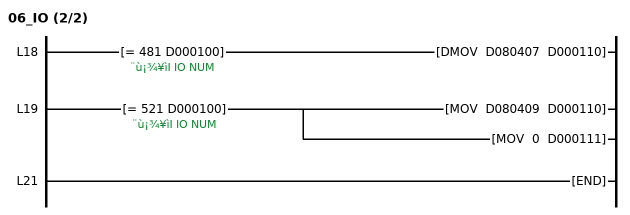
[picture p48: 06_IO rungs L18-L21]
; L18
LOAD=     481 D000100	// ¨ù¡¾¥ìI IO NUM
DMOV      D080407 D000110
; L19
LOAD=     521 D000100	// ¨ù¡¾¥ìI IO NUM
MOV       D080409 D000110
MOV       0 D000111
; L21
END

PROGRAM 07_VACUUM (task: ¨ö¨¬A¥ì CA¡¤I¡¾¡¿¡¤¡Í)

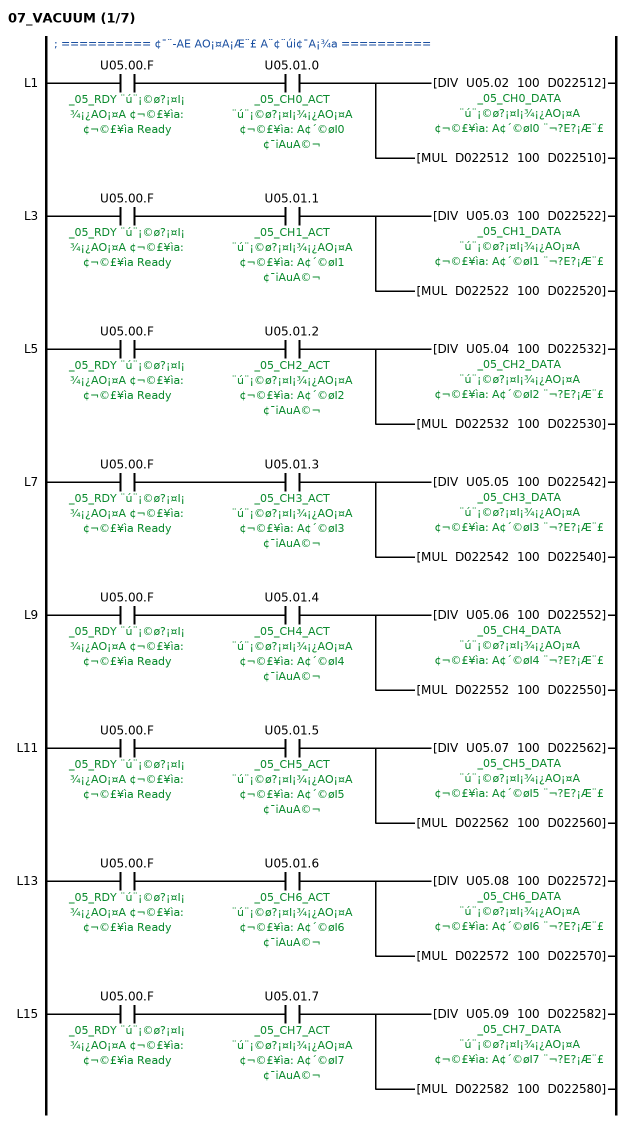
// ========== ¢¯¨­AE AO¡¤A¡Æ¨£ A¨¢¨úi¢¯A¡¾a ==========
; L1
LOAD      U05.00.F	// _05_RDY ¨ú¨¡©ø?¡¤I¡¾¡¿AO¡¤A ¢¬©£¥ìa: ¢¬©£¥ìa Ready
AND       U05.01.0	// _05_CH0_ACT ¨ú¨¡©ø?¡¤I¡¾¡¿AO¡¤A ¢¬©£¥ìa: A¢´©øI0 ¢¯iAuA©¬
DIV       U05.02 100 D022512	// _05_CH0_DATA ¨ú¨¡©ø?¡¤I¡¾¡¿AO¡¤A ¢¬©£¥ìa: A¢´©øI0 ¨¬?E?¡Æ¨£
MUL       D022512 100 D022510
; L3
LOAD      U05.00.F	// _05_RDY ¨ú¨¡©ø?¡¤I¡¾¡¿AO¡¤A ¢¬©£¥ìa: ¢¬©£¥ìa Ready
AND       U05.01.1	// _05_CH1_ACT ¨ú¨¡©ø?¡¤I¡¾¡¿AO¡¤A ¢¬©£¥ìa: A¢´©øI1 ¢¯iAuA©¬
DIV       U05.03 100 D022522	// _05_CH1_DATA ¨ú¨¡©ø?¡¤I¡¾¡¿AO¡¤A ¢¬©£¥ìa: A¢´©øI1 ¨¬?E?¡Æ¨£
MUL       D022522 100 D022520
; L5
LOAD      U05.00.F	// _05_RDY ¨ú¨¡©ø?¡¤I¡¾¡¿AO¡¤A ¢¬©£¥ìa: ¢¬©£¥ìa Ready
AND       U05.01.2	// _05_CH2_ACT ¨ú¨¡©ø?¡¤I¡¾¡¿AO¡¤A ¢¬©£¥ìa: A¢´©øI2 ¢¯iAuA©¬
DIV       U05.04 100 D022532	// _05_CH2_DATA ¨ú¨¡©ø?¡¤I¡¾¡¿AO¡¤A ¢¬©£¥ìa: A¢´©øI2 ¨¬?E?¡Æ¨£
MUL       D022532 100 D022530
; L7
LOAD      U05.00.F	// _05_RDY ¨ú¨¡©ø?¡¤I¡¾¡¿AO¡¤A ¢¬©£¥ìa: ¢¬©£¥ìa Ready
AND       U05.01.3	// _05_CH3_ACT ¨ú¨¡©ø?¡¤I¡¾¡¿AO¡¤A ¢¬©£¥ìa: A¢´©øI3 ¢¯iAuA©¬
DIV       U05.05 100 D022542	// _05_CH3_DATA ¨ú¨¡©ø?¡¤I¡¾¡¿AO¡¤A ¢¬©£¥ìa: A¢´©øI3 ¨¬?E?¡Æ¨£
MUL       D022542 100 D022540
; L9
LOAD      U05.00.F	// _05_RDY ¨ú¨¡©ø?¡¤I¡¾¡¿AO¡¤A ¢¬©£¥ìa: ¢¬©£¥ìa Ready
AND       U05.01.4	// _05_CH4_ACT ¨ú¨¡©ø?¡¤I¡¾¡¿AO¡¤A ¢¬©£¥ìa: A¢´©øI4 ¢¯iAuA©¬
DIV       U05.06 100 D022552	// _05_CH4_DATA ¨ú¨¡©ø?¡¤I¡¾¡¿AO¡¤A ¢¬©£¥ìa: A¢´©øI4 ¨¬?E?¡Æ¨£
MUL       D022552 100 D022550
; L11
LOAD      U05.00.F	// _05_RDY ¨ú¨¡©ø?¡¤I¡¾¡¿AO¡¤A ¢¬©£¥ìa: ¢¬©£¥ìa Ready
AND       U05.01.5	// _05_CH5_ACT ¨ú¨¡©ø?¡¤I¡¾¡¿AO¡¤A ¢¬©£¥ìa: A¢´©øI5 ¢¯iAuA©¬
DIV       U05.07 100 D022562	// _05_CH5_DATA ¨ú¨¡©ø?¡¤I¡¾¡¿AO¡¤A ¢¬©£¥ìa: A¢´©øI5 ¨¬?E?¡Æ¨£
MUL       D022562 100 D022560
; L13
LOAD      U05.00.F	// _05_RDY ¨ú¨¡©ø?¡¤I¡¾¡¿AO¡¤A ¢¬©£¥ìa: ¢¬©£¥ìa Ready
AND       U05.01.6	// _05_CH6_ACT ¨ú¨¡©ø?¡¤I¡¾¡¿AO¡¤A ¢¬©£¥ìa: A¢´©øI6 ¢¯iAuA©¬
DIV       U05.08 100 D022572	// _05_CH6_DATA ¨ú¨¡©ø?¡¤I¡¾¡¿AO¡¤A ¢¬©£¥ìa: A¢´©øI6 ¨¬?E?¡Æ¨£
MUL       D022572 100 D022570
; L15
LOAD      U05.00.F	// _05_RDY ¨ú¨¡©ø?¡¤I¡¾¡¿AO¡¤A ¢¬©£¥ìa: ¢¬©£¥ìa Ready
AND       U05.01.7	// _05_CH7_ACT ¨ú¨¡©ø?¡¤I¡¾¡¿AO¡¤A ¢¬©£¥ìa: A¢´©øI7 ¢¯iAuA©¬
DIV       U05.09 100 D022582	// _05_CH7_DATA ¨ú¨¡©ø?¡¤I¡¾¡¿AO¡¤A ¢¬©£¥ìa: A¢´©øI7 ¨¬?E?¡Æ¨£
MUL       D022582 100 D022580

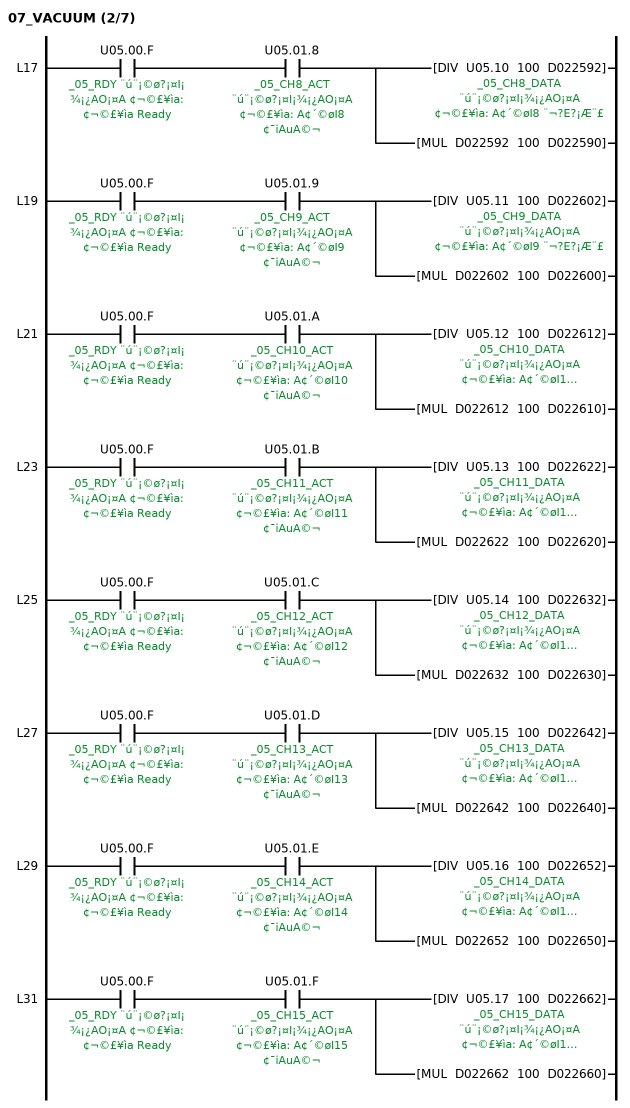
; L17
LOAD      U05.00.F	// _05_RDY ¨ú¨¡©ø?¡¤I¡¾¡¿AO¡¤A ¢¬©£¥ìa: ¢¬©£¥ìa Ready
AND       U05.01.8	// _05_CH8_ACT ¨ú¨¡©ø?¡¤I¡¾¡¿AO¡¤A ¢¬©£¥ìa: A¢´©øI8 ¢¯iAuA©¬
DIV       U05.10 100 D022592	// _05_CH8_DATA ¨ú¨¡©ø?¡¤I¡¾¡¿AO¡¤A ¢¬©£¥ìa: A¢´©øI8 ¨¬?E?¡Æ¨£
MUL       D022592 100 D022590
; L19
LOAD      U05.00.F	// _05_RDY ¨ú¨¡©ø?¡¤I¡¾¡¿AO¡¤A ¢¬©£¥ìa: ¢¬©£¥ìa Ready
AND       U05.01.9	// _05_CH9_ACT ¨ú¨¡©ø?¡¤I¡¾¡¿AO¡¤A ¢¬©£¥ìa: A¢´©øI9 ¢¯iAuA©¬
DIV       U05.11 100 D022602	// _05_CH9_DATA ¨ú¨¡©ø?¡¤I¡¾¡¿AO¡¤A ¢¬©£¥ìa: A¢´©øI9 ¨¬?E?¡Æ¨£
MUL       D022602 100 D022600
; L21
LOAD      U05.00.F	// _05_RDY ¨ú¨¡©ø?¡¤I¡¾¡¿AO¡¤A ¢¬©£¥ìa: ¢¬©£¥ìa Ready
AND       U05.01.A	// _05_CH10_ACT ¨ú¨¡©ø?¡¤I¡¾¡¿AO¡¤A ¢¬©£¥ìa: A¢´©øI10 ¢¯iAuA©¬
DIV       U05.12 100 D022612	// _05_CH10_DATA ¨ú¨¡©ø?¡¤I¡¾¡¿AO¡¤A ¢¬©£¥ìa: A¢´©øI10 ¨¬?E?¡Æ¨£
MUL       D022612 100 D022610
; L23
LOAD      U05.00.F	// _05_RDY ¨ú¨¡©ø?¡¤I¡¾¡¿AO¡¤A ¢¬©£¥ìa: ¢¬©£¥ìa Ready
AND       U05.01.B	// _05_CH11_ACT ¨ú¨¡©ø?¡¤I¡¾¡¿AO¡¤A ¢¬©£¥ìa: A¢´©øI11 ¢¯iAuA©¬
DIV       U05.13 100 D022622	// _05_CH11_DATA ¨ú¨¡©ø?¡¤I¡¾¡¿AO¡¤A ¢¬©£¥ìa: A¢´©øI11 ¨¬?E?¡Æ¨£
MUL       D022622 100 D022620
; L25
LOAD      U05.00.F	// _05_RDY ¨ú¨¡©ø?¡¤I¡¾¡¿AO¡¤A ¢¬©£¥ìa: ¢¬©£¥ìa Ready
AND       U05.01.C	// _05_CH12_ACT ¨ú¨¡©ø?¡¤I¡¾¡¿AO¡¤A ¢¬©£¥ìa: A¢´©øI12 ¢¯iAuA©¬
DIV       U05.14 100 D022632	// _05_CH12_DATA ¨ú¨¡©ø?¡¤I¡¾¡¿AO¡¤A ¢¬©£¥ìa: A¢´©øI12 ¨¬?E?¡Æ¨£
MUL       D022632 100 D022630
; L27
LOAD      U05.00.F	// _05_RDY ¨ú¨¡©ø?¡¤I¡¾¡¿AO¡¤A ¢¬©£¥ìa: ¢¬©£¥ìa Ready
AND       U05.01.D	// _05_CH13_ACT ¨ú¨¡©ø?¡¤I¡¾¡¿AO¡¤A ¢¬©£¥ìa: A¢´©øI13 ¢¯iAuA©¬
DIV       U05.15 100 D022642	// _05_CH13_DATA ¨ú¨¡©ø?¡¤I¡¾¡¿AO¡¤A ¢¬©£¥ìa: A¢´©øI13 ¨¬?E?¡Æ¨£
MUL       D022642 100 D022640
; L29
LOAD      U05.00.F	// _05_RDY ¨ú¨¡©ø?¡¤I¡¾¡¿AO¡¤A ¢¬©£¥ìa: ¢¬©£¥ìa Ready
AND       U05.01.E	// _05_CH14_ACT ¨ú¨¡©ø?¡¤I¡¾¡¿AO¡¤A ¢¬©£¥ìa: A¢´©øI14 ¢¯iAuA©¬
DIV       U05.16 100 D022652	// _05_CH14_DATA ¨ú¨¡©ø?¡¤I¡¾¡¿AO¡¤A ¢¬©£¥ìa: A¢´©øI14 ¨¬?E?¡Æ¨£
MUL       D022652 100 D022650
; L31
LOAD      U05.00.F	// _05_RDY ¨ú¨¡©ø?¡¤I¡¾¡¿AO¡¤A ¢¬©£¥ìa: ¢¬©£¥ìa Ready
AND       U05.01.F	// _05_CH15_ACT ¨ú¨¡©ø?¡¤I¡¾¡¿AO¡¤A ¢¬©£¥ìa: A¢´©øI15 ¢¯iAuA©¬
DIV       U05.17 100 D022662	// _05_CH15_DATA ¨ú¨¡©ø?¡¤I¡¾¡¿AO¡¤A ¢¬©£¥ìa: A¢´©øI15 ¨¬?E?¡Æ¨£
MUL       D022662 100 D022660

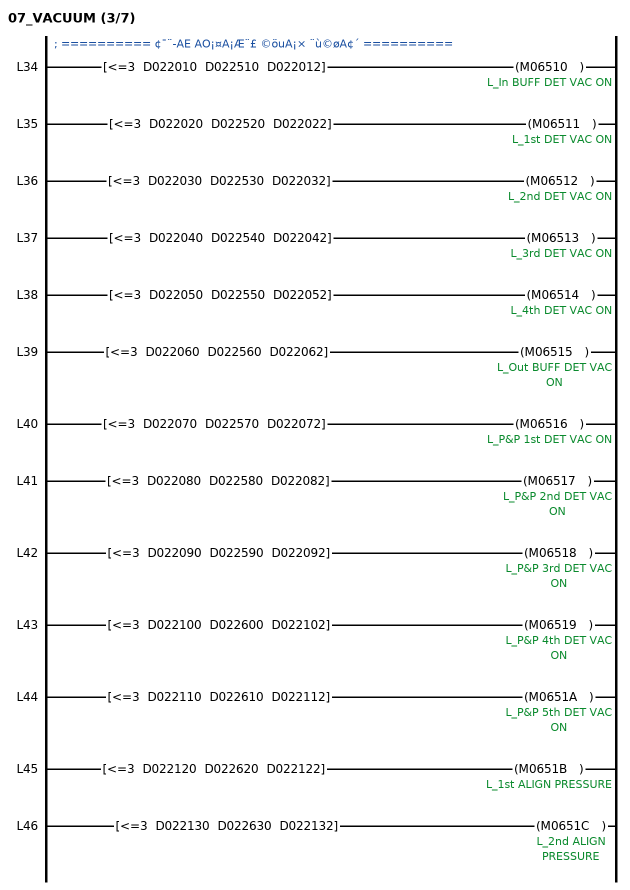
// ========== ¢¯¨­AE AO¡¤A¡Æ¨£ ©öuA¡× ¨ù©øA¢´ ==========
; L34
LOAD<=3   D022010 D022510 D022012
OUT       M06510	// L_In BUFF DET VAC ON
; L35
LOAD<=3   D022020 D022520 D022022
OUT       M06511	// L_1st DET VAC ON
; L36
LOAD<=3   D022030 D022530 D022032
OUT       M06512	// L_2nd DET VAC ON
; L37
LOAD<=3   D022040 D022540 D022042
OUT       M06513	// L_3rd DET VAC ON
; L38
LOAD<=3   D022050 D022550 D022052
OUT       M06514	// L_4th DET VAC ON
; L39
LOAD<=3   D022060 D022560 D022062
OUT       M06515	// L_Out BUFF DET VAC ON
; L40
LOAD<=3   D022070 D022570 D022072
OUT       M06516	// L_P&P 1st DET VAC ON
; L41
LOAD<=3   D022080 D022580 D022082
OUT       M06517	// L_P&P 2nd DET VAC ON
; L42
LOAD<=3   D022090 D022590 D022092
OUT       M06518	// L_P&P 3rd DET VAC ON
; L43
LOAD<=3   D022100 D022600 D022102
OUT       M06519	// L_P&P 4th DET VAC ON
; L44
LOAD<=3   D022110 D022610 D022112
OUT       M0651A	// L_P&P 5th DET VAC ON
; L45
LOAD<=3   D022120 D022620 D022122
OUT       M0651B	// L_1st ALIGN PRESSURE
; L46
LOAD<=3   D022130 D022630 D022132
OUT       M0651C	// L_2nd ALIGN PRESSURE

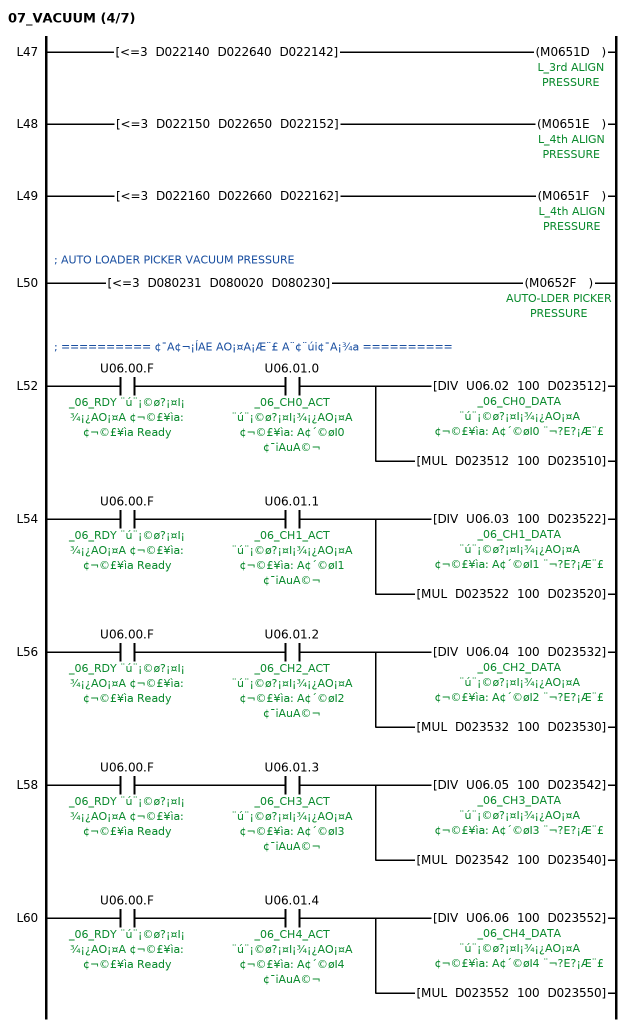
; L47
LOAD<=3   D022140 D022640 D022142
OUT       M0651D	// L_3rd ALIGN PRESSURE
; L48
LOAD<=3   D022150 D022650 D022152
OUT       M0651E	// L_4th ALIGN PRESSURE
; L49
LOAD<=3   D022160 D022660 D022162
OUT       M0651F	// L_4th ALIGN PRESSURE
; L50
LOAD<=3   D080231 D080020 D080230
OUT       M0652F	// AUTO-LDER PICKER PRESSURE
// output comment: AUTO LOADER PICKER VACUUM PRESSURE
// ========== ¢¯A¢¬¡ÍAE AO¡¤A¡Æ¨£ A¨¢¨úi¢¯A¡¾a ==========
; L52
LOAD      U06.00.F	// _06_RDY ¨ú¨¡©ø?¡¤I¡¾¡¿AO¡¤A ¢¬©£¥ìa: ¢¬©£¥ìa Ready
AND       U06.01.0	// _06_CH0_ACT ¨ú¨¡©ø?¡¤I¡¾¡¿AO¡¤A ¢¬©£¥ìa: A¢´©øI0 ¢¯iAuA©¬
DIV       U06.02 100 D023512	// _06_CH0_DATA ¨ú¨¡©ø?¡¤I¡¾¡¿AO¡¤A ¢¬©£¥ìa: A¢´©øI0 ¨¬?E?¡Æ¨£
MUL       D023512 100 D023510
; L54
LOAD      U06.00.F	// _06_RDY ¨ú¨¡©ø?¡¤I¡¾¡¿AO¡¤A ¢¬©£¥ìa: ¢¬©£¥ìa Ready
AND       U06.01.1	// _06_CH1_ACT ¨ú¨¡©ø?¡¤I¡¾¡¿AO¡¤A ¢¬©£¥ìa: A¢´©øI1 ¢¯iAuA©¬
DIV       U06.03 100 D023522	// _06_CH1_DATA ¨ú¨¡©ø?¡¤I¡¾¡¿AO¡¤A ¢¬©£¥ìa: A¢´©øI1 ¨¬?E?¡Æ¨£
MUL       D023522 100 D023520
; L56
LOAD      U06.00.F	// _06_RDY ¨ú¨¡©ø?¡¤I¡¾¡¿AO¡¤A ¢¬©£¥ìa: ¢¬©£¥ìa Ready
AND       U06.01.2	// _06_CH2_ACT ¨ú¨¡©ø?¡¤I¡¾¡¿AO¡¤A ¢¬©£¥ìa: A¢´©øI2 ¢¯iAuA©¬
DIV       U06.04 100 D023532	// _06_CH2_DATA ¨ú¨¡©ø?¡¤I¡¾¡¿AO¡¤A ¢¬©£¥ìa: A¢´©øI2 ¨¬?E?¡Æ¨£
MUL       D023532 100 D023530
; L58
LOAD      U06.00.F	// _06_RDY ¨ú¨¡©ø?¡¤I¡¾¡¿AO¡¤A ¢¬©£¥ìa: ¢¬©£¥ìa Ready
AND       U06.01.3	// _06_CH3_ACT ¨ú¨¡©ø?¡¤I¡¾¡¿AO¡¤A ¢¬©£¥ìa: A¢´©øI3 ¢¯iAuA©¬
DIV       U06.05 100 D023542	// _06_CH3_DATA ¨ú¨¡©ø?¡¤I¡¾¡¿AO¡¤A ¢¬©£¥ìa: A¢´©øI3 ¨¬?E?¡Æ¨£
MUL       D023542 100 D023540
; L60
LOAD      U06.00.F	// _06_RDY ¨ú¨¡©ø?¡¤I¡¾¡¿AO¡¤A ¢¬©£¥ìa: ¢¬©£¥ìa Ready
AND       U06.01.4	// _06_CH4_ACT ¨ú¨¡©ø?¡¤I¡¾¡¿AO¡¤A ¢¬©£¥ìa: A¢´©øI4 ¢¯iAuA©¬
DIV       U06.06 100 D023552	// _06_CH4_DATA ¨ú¨¡©ø?¡¤I¡¾¡¿AO¡¤A ¢¬©£¥ìa: A¢´©øI4 ¨¬?E?¡Æ¨£
MUL       D023552 100 D023550

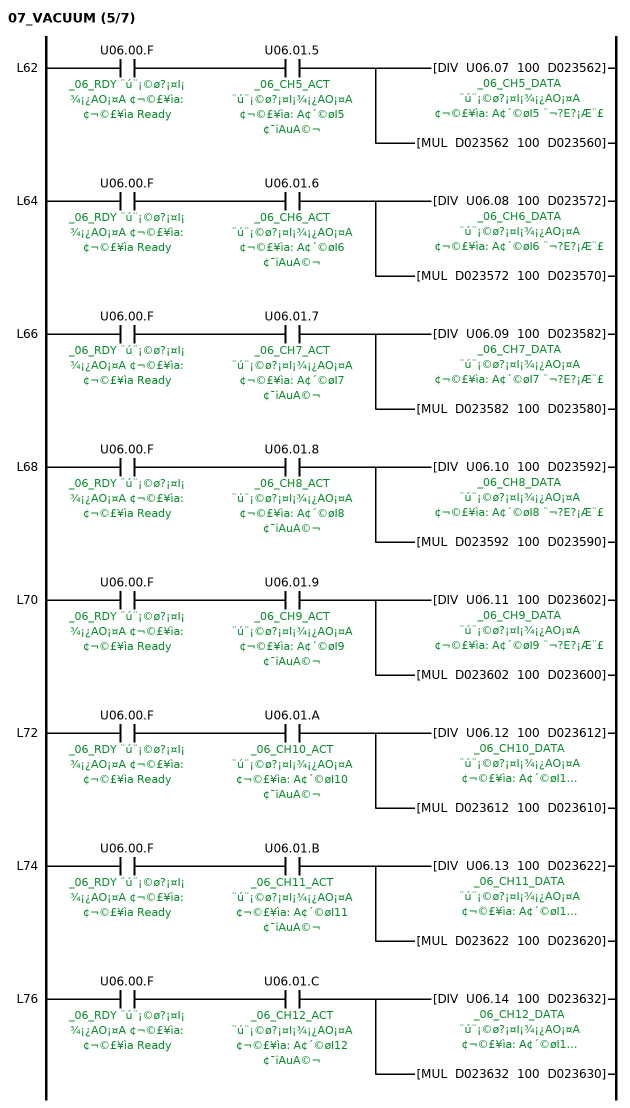
; L62
LOAD      U06.00.F	// _06_RDY ¨ú¨¡©ø?¡¤I¡¾¡¿AO¡¤A ¢¬©£¥ìa: ¢¬©£¥ìa Ready
AND       U06.01.5	// _06_CH5_ACT ¨ú¨¡©ø?¡¤I¡¾¡¿AO¡¤A ¢¬©£¥ìa: A¢´©øI5 ¢¯iAuA©¬
DIV       U06.07 100 D023562	// _06_CH5_DATA ¨ú¨¡©ø?¡¤I¡¾¡¿AO¡¤A ¢¬©£¥ìa: A¢´©øI5 ¨¬?E?¡Æ¨£
MUL       D023562 100 D023560
; L64
LOAD      U06.00.F	// _06_RDY ¨ú¨¡©ø?¡¤I¡¾¡¿AO¡¤A ¢¬©£¥ìa: ¢¬©£¥ìa Ready
AND       U06.01.6	// _06_CH6_ACT ¨ú¨¡©ø?¡¤I¡¾¡¿AO¡¤A ¢¬©£¥ìa: A¢´©øI6 ¢¯iAuA©¬
DIV       U06.08 100 D023572	// _06_CH6_DATA ¨ú¨¡©ø?¡¤I¡¾¡¿AO¡¤A ¢¬©£¥ìa: A¢´©øI6 ¨¬?E?¡Æ¨£
MUL       D023572 100 D023570
; L66
LOAD      U06.00.F	// _06_RDY ¨ú¨¡©ø?¡¤I¡¾¡¿AO¡¤A ¢¬©£¥ìa: ¢¬©£¥ìa Ready
AND       U06.01.7	// _06_CH7_ACT ¨ú¨¡©ø?¡¤I¡¾¡¿AO¡¤A ¢¬©£¥ìa: A¢´©øI7 ¢¯iAuA©¬
DIV       U06.09 100 D023582	// _06_CH7_DATA ¨ú¨¡©ø?¡¤I¡¾¡¿AO¡¤A ¢¬©£¥ìa: A¢´©øI7 ¨¬?E?¡Æ¨£
MUL       D023582 100 D023580
; L68
LOAD      U06.00.F	// _06_RDY ¨ú¨¡©ø?¡¤I¡¾¡¿AO¡¤A ¢¬©£¥ìa: ¢¬©£¥ìa Ready
AND       U06.01.8	// _06_CH8_ACT ¨ú¨¡©ø?¡¤I¡¾¡¿AO¡¤A ¢¬©£¥ìa: A¢´©øI8 ¢¯iAuA©¬
DIV       U06.10 100 D023592	// _06_CH8_DATA ¨ú¨¡©ø?¡¤I¡¾¡¿AO¡¤A ¢¬©£¥ìa: A¢´©øI8 ¨¬?E?¡Æ¨£
MUL       D023592 100 D023590
; L70
LOAD      U06.00.F	// _06_RDY ¨ú¨¡©ø?¡¤I¡¾¡¿AO¡¤A ¢¬©£¥ìa: ¢¬©£¥ìa Ready
AND       U06.01.9	// _06_CH9_ACT ¨ú¨¡©ø?¡¤I¡¾¡¿AO¡¤A ¢¬©£¥ìa: A¢´©øI9 ¢¯iAuA©¬
DIV       U06.11 100 D023602	// _06_CH9_DATA ¨ú¨¡©ø?¡¤I¡¾¡¿AO¡¤A ¢¬©£¥ìa: A¢´©øI9 ¨¬?E?¡Æ¨£
MUL       D023602 100 D023600
; L72
LOAD      U06.00.F	// _06_RDY ¨ú¨¡©ø?¡¤I¡¾¡¿AO¡¤A ¢¬©£¥ìa: ¢¬©£¥ìa Ready
AND       U06.01.A	// _06_CH10_ACT ¨ú¨¡©ø?¡¤I¡¾¡¿AO¡¤A ¢¬©£¥ìa: A¢´©øI10 ¢¯iAuA©¬
DIV       U06.12 100 D023612	// _06_CH10_DATA ¨ú¨¡©ø?¡¤I¡¾¡¿AO¡¤A ¢¬©£¥ìa: A¢´©øI10 ¨¬?E?¡Æ¨£
MUL       D023612 100 D023610
; L74
LOAD      U06.00.F	// _06_RDY ¨ú¨¡©ø?¡¤I¡¾¡¿AO¡¤A ¢¬©£¥ìa: ¢¬©£¥ìa Ready
AND       U06.01.B	// _06_CH11_ACT ¨ú¨¡©ø?¡¤I¡¾¡¿AO¡¤A ¢¬©£¥ìa: A¢´©øI11 ¢¯iAuA©¬
DIV       U06.13 100 D023622	// _06_CH11_DATA ¨ú¨¡©ø?¡¤I¡¾¡¿AO¡¤A ¢¬©£¥ìa: A¢´©øI11 ¨¬?E?¡Æ¨£
MUL       D023622 100 D023620
; L76
LOAD      U06.00.F	// _06_RDY ¨ú¨¡©ø?¡¤I¡¾¡¿AO¡¤A ¢¬©£¥ìa: ¢¬©£¥ìa Ready
AND       U06.01.C	// _06_CH12_ACT ¨ú¨¡©ø?¡¤I¡¾¡¿AO¡¤A ¢¬©£¥ìa: A¢´©øI12 ¢¯iAuA©¬
DIV       U06.14 100 D023632	// _06_CH12_DATA ¨ú¨¡©ø?¡¤I¡¾¡¿AO¡¤A ¢¬©£¥ìa: A¢´©øI12 ¨¬?E?¡Æ¨£
MUL       D023632 100 D023630

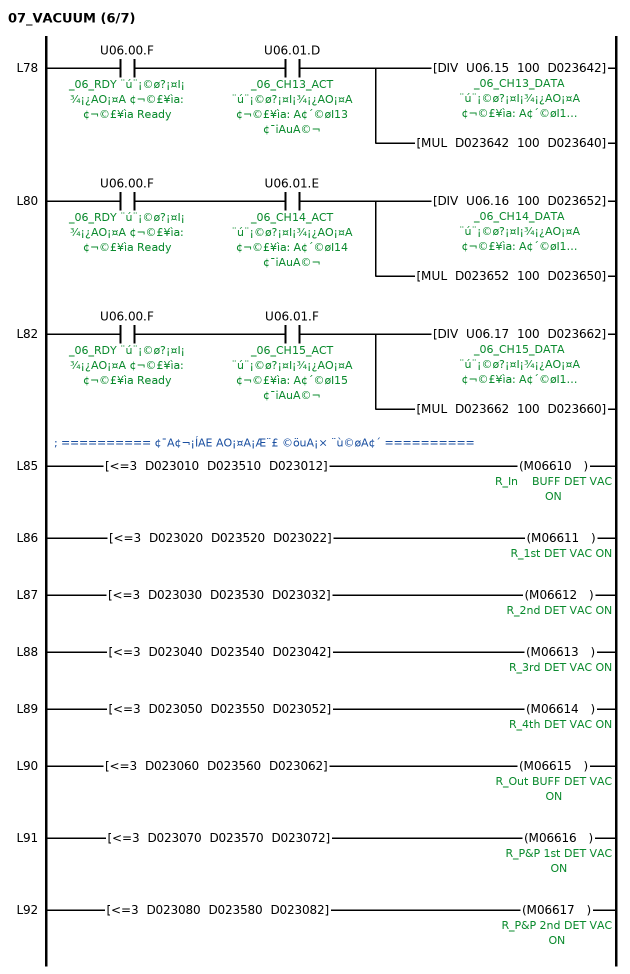
; L78
LOAD      U06.00.F	// _06_RDY ¨ú¨¡©ø?¡¤I¡¾¡¿AO¡¤A ¢¬©£¥ìa: ¢¬©£¥ìa Ready
AND       U06.01.D	// _06_CH13_ACT ¨ú¨¡©ø?¡¤I¡¾¡¿AO¡¤A ¢¬©£¥ìa: A¢´©øI13 ¢¯iAuA©¬
DIV       U06.15 100 D023642	// _06_CH13_DATA ¨ú¨¡©ø?¡¤I¡¾¡¿AO¡¤A ¢¬©£¥ìa: A¢´©øI13 ¨¬?E?¡Æ¨£
MUL       D023642 100 D023640
; L80
LOAD      U06.00.F	// _06_RDY ¨ú¨¡©ø?¡¤I¡¾¡¿AO¡¤A ¢¬©£¥ìa: ¢¬©£¥ìa Ready
AND       U06.01.E	// _06_CH14_ACT ¨ú¨¡©ø?¡¤I¡¾¡¿AO¡¤A ¢¬©£¥ìa: A¢´©øI14 ¢¯iAuA©¬
DIV       U06.16 100 D023652	// _06_CH14_DATA ¨ú¨¡©ø?¡¤I¡¾¡¿AO¡¤A ¢¬©£¥ìa: A¢´©øI14 ¨¬?E?¡Æ¨£
MUL       D023652 100 D023650
; L82
LOAD      U06.00.F	// _06_RDY ¨ú¨¡©ø?¡¤I¡¾¡¿AO¡¤A ¢¬©£¥ìa: ¢¬©£¥ìa Ready
AND       U06.01.F	// _06_CH15_ACT ¨ú¨¡©ø?¡¤I¡¾¡¿AO¡¤A ¢¬©£¥ìa: A¢´©øI15 ¢¯iAuA©¬
DIV       U06.17 100 D023662	// _06_CH15_DATA ¨ú¨¡©ø?¡¤I¡¾¡¿AO¡¤A ¢¬©£¥ìa: A¢´©øI15 ¨¬?E?¡Æ¨£
MUL       D023662 100 D023660
// ========== ¢¯A¢¬¡ÍAE AO¡¤A¡Æ¨£ ©öuA¡× ¨ù©øA¢´ ==========
; L85
LOAD<=3   D023010 D023510 D023012
OUT       M06610	// R_In    BUFF DET VAC ON
; L86
LOAD<=3   D023020 D023520 D023022
OUT       M06611	// R_1st DET VAC ON
; L87
LOAD<=3   D023030 D023530 D023032
OUT       M06612	// R_2nd DET VAC ON
; L88
LOAD<=3   D023040 D023540 D023042
OUT       M06613	// R_3rd DET VAC ON
; L89
LOAD<=3   D023050 D023550 D023052
OUT       M06614	// R_4th DET VAC ON
; L90
LOAD<=3   D023060 D023560 D023062
OUT       M06615	// R_Out BUFF DET VAC ON
; L91
LOAD<=3   D023070 D023570 D023072
OUT       M06616	// R_P&P 1st DET VAC ON
; L92
LOAD<=3   D023080 D023580 D023082
OUT       M06617	// R_P&P 2nd DET VAC ON

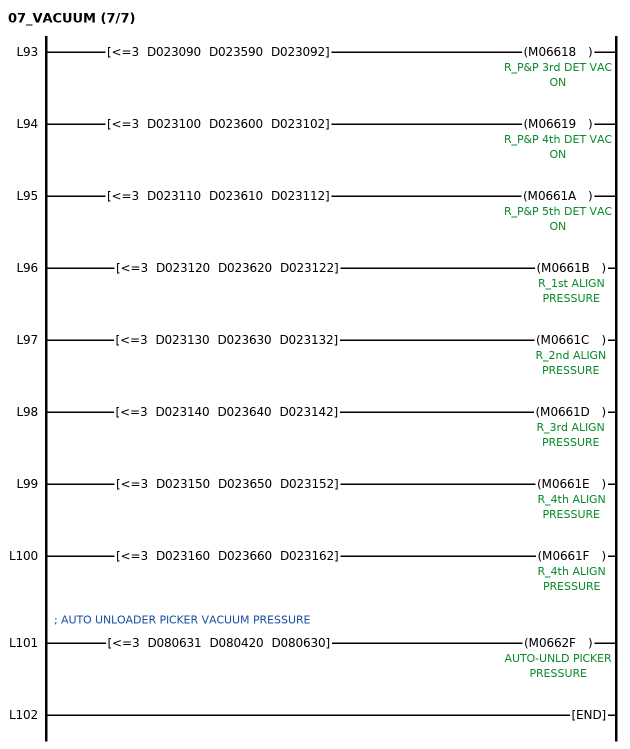
; L93
LOAD<=3   D023090 D023590 D023092
OUT       M06618	// R_P&P 3rd DET VAC ON
; L94
LOAD<=3   D023100 D023600 D023102
OUT       M06619	// R_P&P 4th DET VAC ON
; L95
LOAD<=3   D023110 D023610 D023112
OUT       M0661A	// R_P&P 5th DET VAC ON
; L96
LOAD<=3   D023120 D023620 D023122
OUT       M0661B	// R_1st ALIGN PRESSURE
; L97
LOAD<=3   D023130 D023630 D023132
OUT       M0661C	// R_2nd ALIGN PRESSURE
; L98
LOAD<=3   D023140 D023640 D023142
OUT       M0661D	// R_3rd ALIGN PRESSURE
; L99
LOAD<=3   D023150 D023650 D023152
OUT       M0661E	// R_4th ALIGN PRESSURE
; L100
LOAD<=3   D023160 D023660 D023162
OUT       M0661F	// R_4th ALIGN PRESSURE
; L101
LOAD<=3   D080631 D080420 D080630
OUT       M0662F	// AUTO-UNLD PICKER PRESSURE
// output comment: AUTO UNLOADER PICKER VACUUM PRESSURE
; L102
END

PROGRAM 11_L_1st_MAND (task: ¨ö¨¬A¥ì CA¡¤I¡¾¡¿¡¤¡Í)

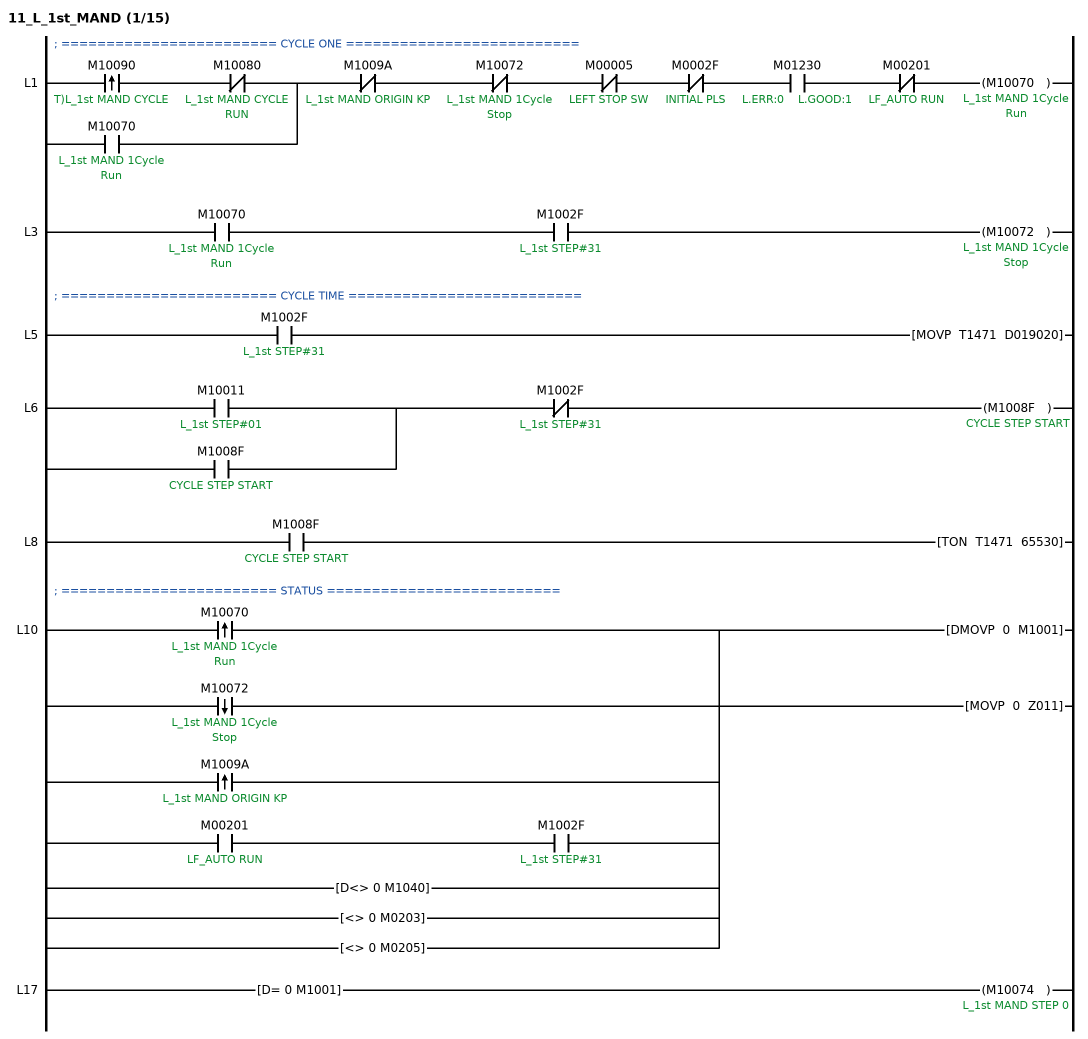
// ======================== CYCLE ONE ==========================
; L1
LOADP     M10090	// T)L_1st MAND CYCLE
AND NOT   M10080	// L_1st MAND CYCLE RUN
OR        M10070	// L_1st MAND 1Cycle Run
AND NOT   M1009A	// L_1st MAND ORIGIN KP
AND NOT   M10072	// L_1st MAND 1Cycle Stop
AND NOT   M00005	// LEFT STOP SW
AND NOT   M0002F	// INITIAL PLS
AND       M01230	// L.ERR:0    L.GOOD:1
AND NOT   M00201	// LF_AUTO RUN
OUT       M10070	// L_1st MAND 1Cycle Run
; L3
LOAD      M10070	// L_1st MAND 1Cycle Run
AND       M1002F	// L_1st STEP#31
OUT       M10072	// L_1st MAND 1Cycle Stop
// ======================== CYCLE TIME ==========================
; L5
LOAD      M1002F	// L_1st STEP#31
MOVP      T1471 D019020
; L6
LOAD      M10011	// L_1st STEP#01
OR        M1008F	// CYCLE STEP START
AND NOT   M1002F	// L_1st STEP#31
OUT       M1008F	// CYCLE STEP START
; L8
LOAD      M1008F	// CYCLE STEP START
TON       T1471 65530
// ======================== STATUS ==========================
; L10
LOADP     M10070	// L_1st MAND 1Cycle Run
ORN       M10072	// L_1st MAND 1Cycle Stop
ORP       M1009A	// L_1st MAND ORIGIN KP
LOAD      M00201	// LF_AUTO RUN
AND       M1002F	// L_1st STEP#31
OR LOAD
ORD<>     0 M1040
OR<>      0 M0203
OR<>      0 M0205
DMOVP     0 M1001
MOVP      0 Z011
; L17
LOADD=    0 M1001
OUT       M10074	// L_1st MAND STEP 0

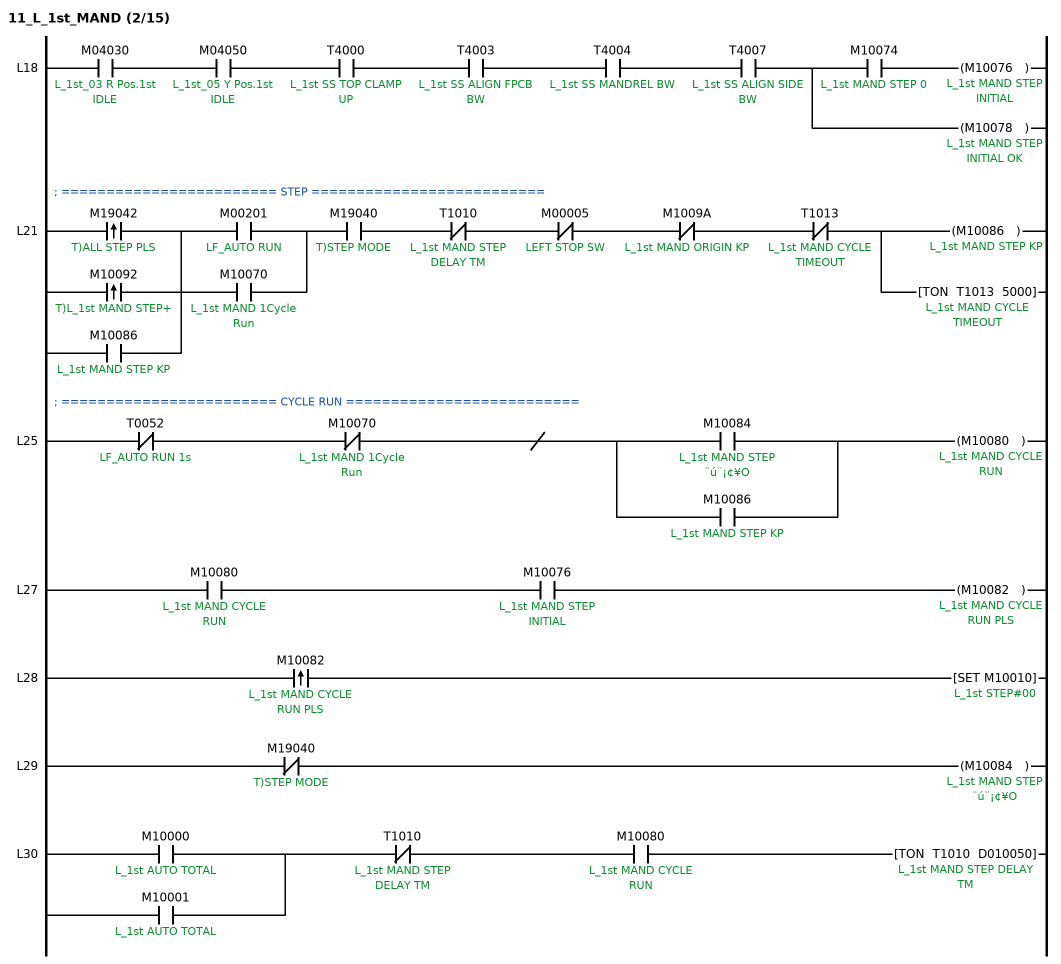
; L18
LOAD      M04030	// L_1st_03 R Pos.1st IDLE
AND       M04050	// L_1st_05 Y Pos.1st IDLE
AND       T4000	// L_1st SS TOP CLAMP    UP
AND       T4003	// L_1st SS ALIGN FPCB BW
AND       T4004	// L_1st SS MANDREL BW
AND       T4007	// L_1st SS ALIGN SIDE BW
MPUSH
AND       M10074	// L_1st MAND STEP 0
OUT       M10076	// L_1st MAND STEP INITIAL
MPOP
OUT       M10078	// L_1st MAND STEP INITIAL OK
// ======================== STEP ==========================
; L21
LOADP     M19042	// T)ALL STEP PLS
ORP       M10092	// T)L_1st MAND STEP+
OR        M10086	// L_1st MAND STEP KP
LOAD      M00201	// LF_AUTO RUN
OR        M10070	// L_1st MAND 1Cycle Run
AND LOAD
AND       M19040	// T)STEP MODE
AND NOT   T1010	// L_1st MAND STEP DELAY TM
AND NOT   M00005	// LEFT STOP SW
AND NOT   M1009A	// L_1st MAND ORIGIN KP
AND NOT   T1013	// L_1st MAND CYCLE TIMEOUT
OUT       M10086	// L_1st MAND STEP KP
TON       T1013 5000	// L_1st MAND CYCLE TIMEOUT
// ======================== CYCLE RUN ==========================
; L25
LOAD NOT  T0052	// LF_AUTO RUN 1s
AND NOT   M10070	// L_1st MAND 1Cycle Run
NOT
LOAD      M10084	// L_1st MAND STEP ¨ú¨¡¢¥O
OR        M10086	// L_1st MAND STEP KP
AND LOAD
OUT       M10080	// L_1st MAND CYCLE RUN
; L27
LOAD      M10080	// L_1st MAND CYCLE RUN
AND       M10076	// L_1st MAND STEP INITIAL
OUT       M10082	// L_1st MAND CYCLE RUN PLS
; L28
LOADP     M10082	// L_1st MAND CYCLE RUN PLS
SET       M10010	// L_1st STEP#00
; L29
LOAD NOT  M19040	// T)STEP MODE
OUT       M10084	// L_1st MAND STEP ¨ú¨¡¢¥O
; L30
LOAD      M10000	// L_1st AUTO TOTAL
OR        M10001	// L_1st AUTO TOTAL
AND NOT   T1010	// L_1st MAND STEP DELAY TM
AND       M10080	// L_1st MAND CYCLE RUN
TON       T1010 D010050	// L_1st MAND STEP DELAY TM

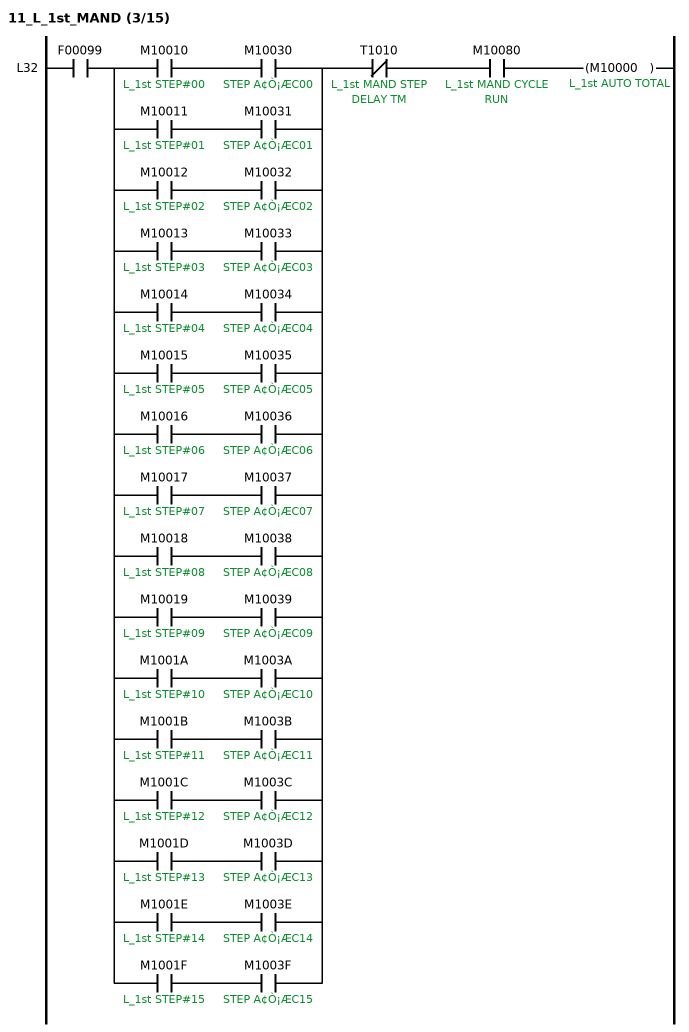
; L32
LOAD      F00099
LOAD      M10010	// L_1st STEP#00
AND       M10030	// STEP A¢Ò¡ÆC00
LOAD      M10011	// L_1st STEP#01
AND       M10031	// STEP A¢Ò¡ÆC01
OR LOAD
LOAD      M10012	// L_1st STEP#02
AND       M10032	// STEP A¢Ò¡ÆC02
OR LOAD
LOAD      M10013	// L_1st STEP#03
AND       M10033	// STEP A¢Ò¡ÆC03
OR LOAD
LOAD      M10014	// L_1st STEP#04
AND       M10034	// STEP A¢Ò¡ÆC04
OR LOAD
LOAD      M10015	// L_1st STEP#05
AND       M10035	// STEP A¢Ò¡ÆC05
OR LOAD
LOAD      M10016	// L_1st STEP#06
AND       M10036	// STEP A¢Ò¡ÆC06
OR LOAD
LOAD      M10017	// L_1st STEP#07
AND       M10037	// STEP A¢Ò¡ÆC07
OR LOAD
LOAD      M10018	// L_1st STEP#08
AND       M10038	// STEP A¢Ò¡ÆC08
OR LOAD
LOAD      M10019	// L_1st STEP#09
AND       M10039	// STEP A¢Ò¡ÆC09
OR LOAD
LOAD      M1001A	// L_1st STEP#10
AND       M1003A	// STEP A¢Ò¡ÆC10
OR LOAD
LOAD      M1001B	// L_1st STEP#11
AND       M1003B	// STEP A¢Ò¡ÆC11
OR LOAD
LOAD      M1001C	// L_1st STEP#12
AND       M1003C	// STEP A¢Ò¡ÆC12
OR LOAD
LOAD      M1001D	// L_1st STEP#13
AND       M1003D	// STEP A¢Ò¡ÆC13
OR LOAD
LOAD      M1001E	// L_1st STEP#14
AND       M1003E	// STEP A¢Ò¡ÆC14
OR LOAD
LOAD      M1001F	// L_1st STEP#15
AND       M1003F	// STEP A¢Ò¡ÆC15
OR LOAD
AND LOAD
AND NOT   T1010	// L_1st MAND STEP DELAY TM
AND       M10080	// L_1st MAND CYCLE RUN
OUT       M10000	// L_1st AUTO TOTAL

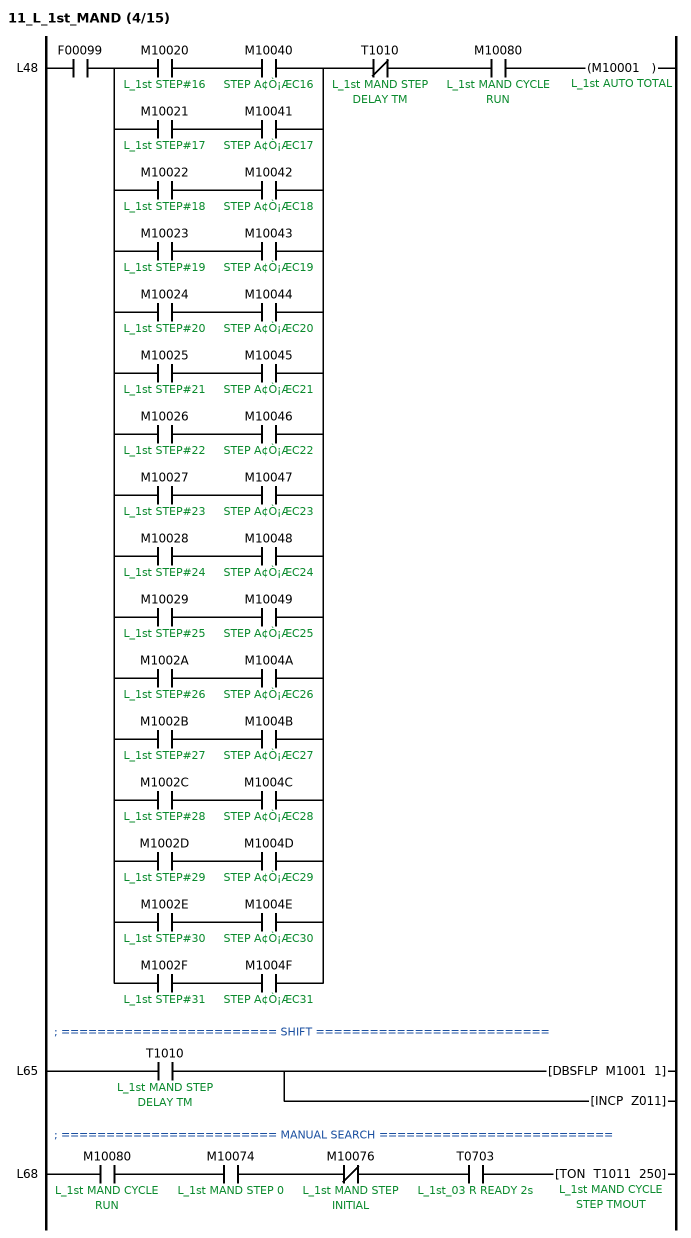
; L48
LOAD      F00099
LOAD      M10020	// L_1st STEP#16
AND       M10040	// STEP A¢Ò¡ÆC16
LOAD      M10021	// L_1st STEP#17
AND       M10041	// STEP A¢Ò¡ÆC17
OR LOAD
LOAD      M10022	// L_1st STEP#18
AND       M10042	// STEP A¢Ò¡ÆC18
OR LOAD
LOAD      M10023	// L_1st STEP#19
AND       M10043	// STEP A¢Ò¡ÆC19
OR LOAD
LOAD      M10024	// L_1st STEP#20
AND       M10044	// STEP A¢Ò¡ÆC20
OR LOAD
LOAD      M10025	// L_1st STEP#21
AND       M10045	// STEP A¢Ò¡ÆC21
OR LOAD
LOAD      M10026	// L_1st STEP#22
AND       M10046	// STEP A¢Ò¡ÆC22
OR LOAD
LOAD      M10027	// L_1st STEP#23
AND       M10047	// STEP A¢Ò¡ÆC23
OR LOAD
LOAD      M10028	// L_1st STEP#24
AND       M10048	// STEP A¢Ò¡ÆC24
OR LOAD
LOAD      M10029	// L_1st STEP#25
AND       M10049	// STEP A¢Ò¡ÆC25
OR LOAD
LOAD      M1002A	// L_1st STEP#26
AND       M1004A	// STEP A¢Ò¡ÆC26
OR LOAD
LOAD      M1002B	// L_1st STEP#27
AND       M1004B	// STEP A¢Ò¡ÆC27
OR LOAD
LOAD      M1002C	// L_1st STEP#28
AND       M1004C	// STEP A¢Ò¡ÆC28
OR LOAD
LOAD      M1002D	// L_1st STEP#29
AND       M1004D	// STEP A¢Ò¡ÆC29
OR LOAD
LOAD      M1002E	// L_1st STEP#30
AND       M1004E	// STEP A¢Ò¡ÆC30
OR LOAD
LOAD      M1002F	// L_1st STEP#31
AND       M1004F	// STEP A¢Ò¡ÆC31
OR LOAD
AND LOAD
AND NOT   T1010	// L_1st MAND STEP DELAY TM
AND       M10080	// L_1st MAND CYCLE RUN
OUT       M10001	// L_1st AUTO TOTAL
// ======================== SHIFT ==========================
; L65
LOAD      T1010	// L_1st MAND STEP DELAY TM
DBSFLP    M1001 1
INCP      Z011
// ======================== MANUAL SEARCH ==========================
; L68
LOAD      M10080	// L_1st MAND CYCLE RUN
AND       M10074	// L_1st MAND STEP 0
AND NOT   M10076	// L_1st MAND STEP INITIAL
AND       T0703	// L_1st_03 R READY 2s
TON       T1011 250	// L_1st MAND CYCLE STEP TMOUT

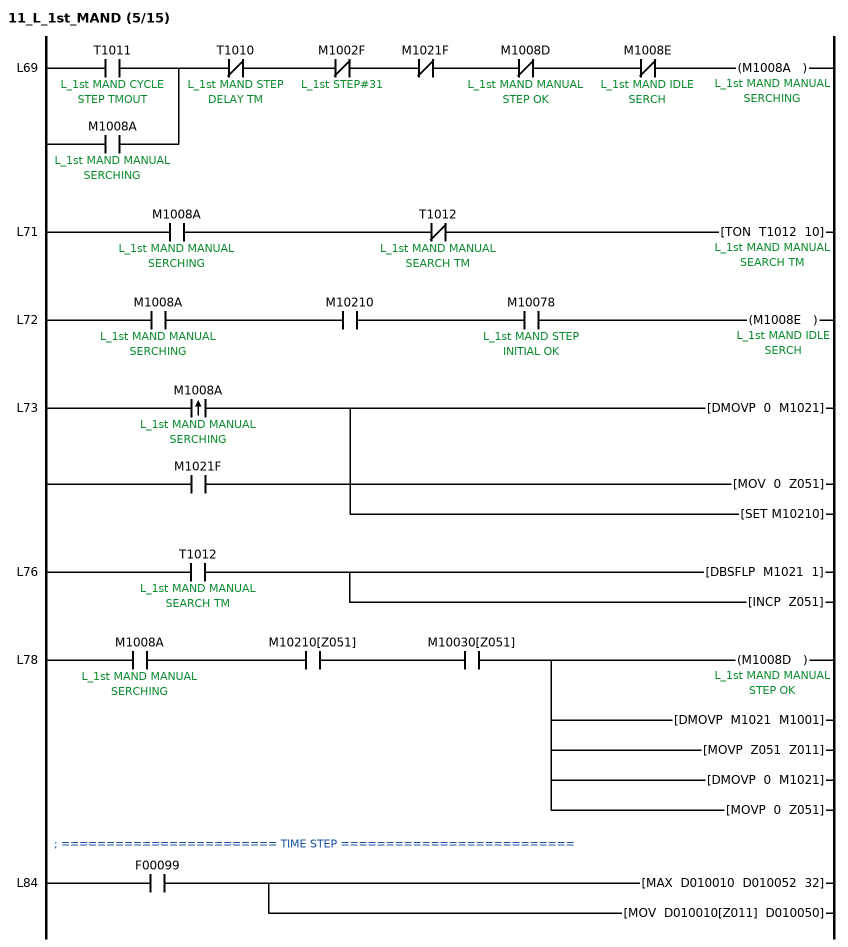
; L69
LOAD      T1011	// L_1st MAND CYCLE STEP TMOUT
OR        M1008A	// L_1st MAND MANUAL SERCHING
AND NOT   T1010	// L_1st MAND STEP DELAY TM
AND NOT   M1002F	// L_1st STEP#31
AND NOT   M1021F
AND NOT   M1008D	// L_1st MAND MANUAL STEP OK
AND NOT   M1008E	// L_1st MAND IDLE SERCH
OUT       M1008A	// L_1st MAND MANUAL SERCHING
; L71
LOAD      M1008A	// L_1st MAND MANUAL SERCHING
AND NOT   T1012	// L_1st MAND MANUAL SEARCH TM
TON       T1012 10	// L_1st MAND MANUAL SEARCH TM
; L72
LOAD      M1008A	// L_1st MAND MANUAL SERCHING
AND       M10210
AND       M10078	// L_1st MAND STEP INITIAL OK
OUT       M1008E	// L_1st MAND IDLE SERCH
; L73
LOADP     M1008A	// L_1st MAND MANUAL SERCHING
OR        M1021F
DMOVP     0 M1021
MOV       0 Z051
SET       M10210
; L76
LOAD      T1012	// L_1st MAND MANUAL SEARCH TM
DBSFLP    M1021 1
INCP      Z051
; L78
LOAD      M1008A	// L_1st MAND MANUAL SERCHING
AND       M10210[Z051]
AND       M10030[Z051]
OUT       M1008D	// L_1st MAND MANUAL STEP OK
DMOVP     M1021 M1001
MOVP      Z051 Z011
DMOVP     0 M1021
MOVP      0 Z051
// ======================== TIME STEP ==========================
; L84
LOAD      F00099
MAX       D010010 D010052 32
MOV       D010010[Z011] D010050

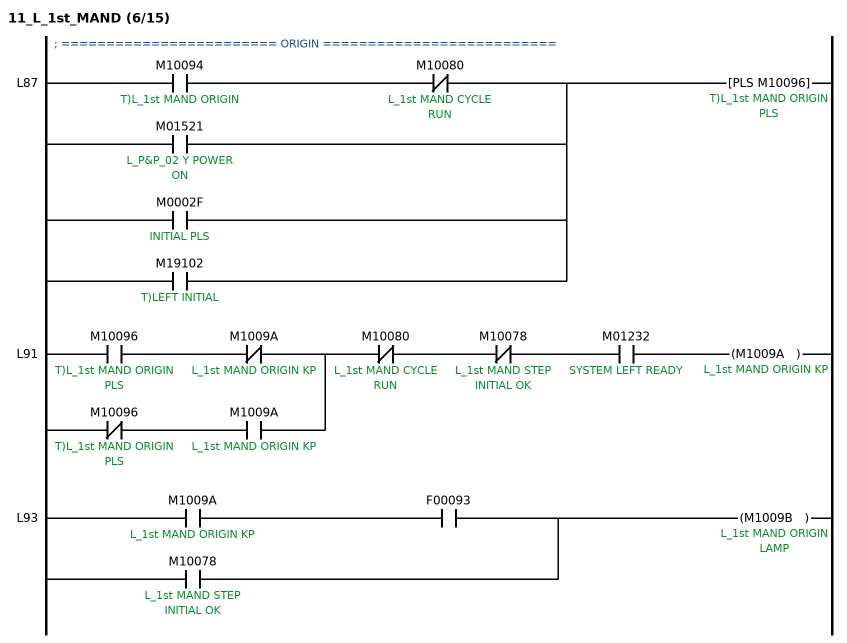
// ======================== ORIGIN ==========================
; L87
LOAD      M10094	// T)L_1st MAND ORIGIN
AND NOT   M10080	// L_1st MAND CYCLE RUN
OR        M01521	// L_P&P_02 Y POWER ON
OR        M0002F	// INITIAL PLS
OR        M19102	// T)LEFT INITIAL
OUTP      M10096	// T)L_1st MAND ORIGIN PLS
; L91
LOAD      M10096	// T)L_1st MAND ORIGIN PLS
AND NOT   M1009A	// L_1st MAND ORIGIN KP
LOAD NOT  M10096	// T)L_1st MAND ORIGIN PLS
AND       M1009A	// L_1st MAND ORIGIN KP
OR LOAD
AND NOT   M10080	// L_1st MAND CYCLE RUN
AND NOT   M10078	// L_1st MAND STEP INITIAL OK
AND       M01232	// SYSTEM LEFT READY
OUT       M1009A	// L_1st MAND ORIGIN KP
; L93
LOAD      M1009A	// L_1st MAND ORIGIN KP
AND       F00093
OR        M10078	// L_1st MAND STEP INITIAL OK
OUT       M1009B	// L_1st MAND ORIGIN LAMP

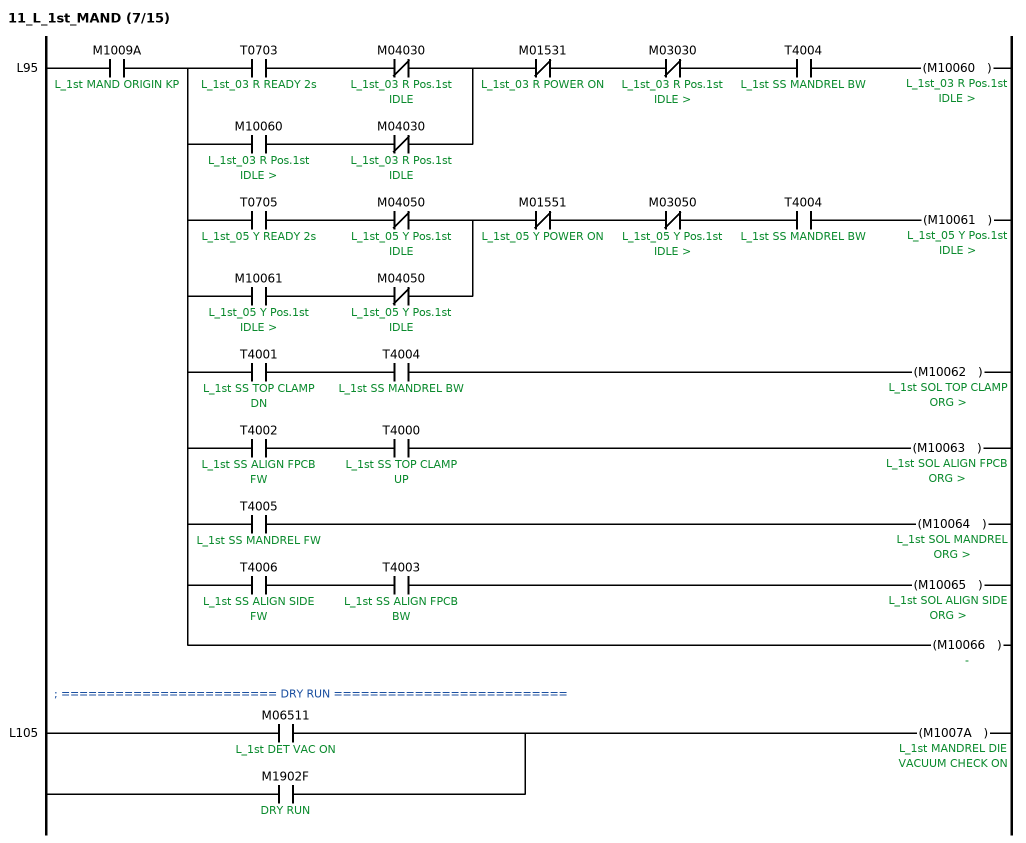
; L95
LOAD      M1009A	// L_1st MAND ORIGIN KP
MPUSH
LOAD      T0703	// L_1st_03 R READY 2s
AND NOT   M04030	// L_1st_03 R Pos.1st IDLE
LOAD      M10060	// L_1st_03 R Pos.1st IDLE >
AND NOT   M04030	// L_1st_03 R Pos.1st IDLE
OR LOAD
AND LOAD
AND NOT   M01531	// L_1st_03 R POWER ON
AND NOT   M03030	// L_1st_03 R Pos.1st IDLE >
AND       T4004	// L_1st SS MANDREL BW
OUT       M10060	// L_1st_03 R Pos.1st IDLE >
MLOAD
LOAD      T0705	// L_1st_05 Y READY 2s
AND NOT   M04050	// L_1st_05 Y Pos.1st IDLE
LOAD      M10061	// L_1st_05 Y Pos.1st IDLE >
AND NOT   M04050	// L_1st_05 Y Pos.1st IDLE
OR LOAD
AND LOAD
AND NOT   M01551	// L_1st_05 Y POWER ON
AND NOT   M03050	// L_1st_05 Y Pos.1st IDLE >
AND       T4004	// L_1st SS MANDREL BW
OUT       M10061	// L_1st_05 Y Pos.1st IDLE >
MLOAD
AND       T4001	// L_1st SS TOP CLAMP    DN
AND       T4004	// L_1st SS MANDREL BW
OUT       M10062	// L_1st SOL TOP CLAMP ORG >
MLOAD
AND       T4002	// L_1st SS ALIGN FPCB FW
AND       T4000	// L_1st SS TOP CLAMP    UP
OUT       M10063	// L_1st SOL ALIGN FPCB ORG >
MLOAD
AND       T4005	// L_1st SS MANDREL FW
OUT       M10064	// L_1st SOL MANDREL ORG >
MLOAD
AND       T4006	// L_1st SS ALIGN SIDE FW
AND       T4003	// L_1st SS ALIGN FPCB BW
OUT       M10065	// L_1st SOL ALIGN SIDE ORG >
MPOP
OUT       M10066	// -
// ======================== DRY RUN ==========================
; L105
LOAD      M06511	// L_1st DET VAC ON
OR        M1902F	// DRY RUN
OUT       M1007A	// L_1st MANDREL DIE VACUUM CHECK ON

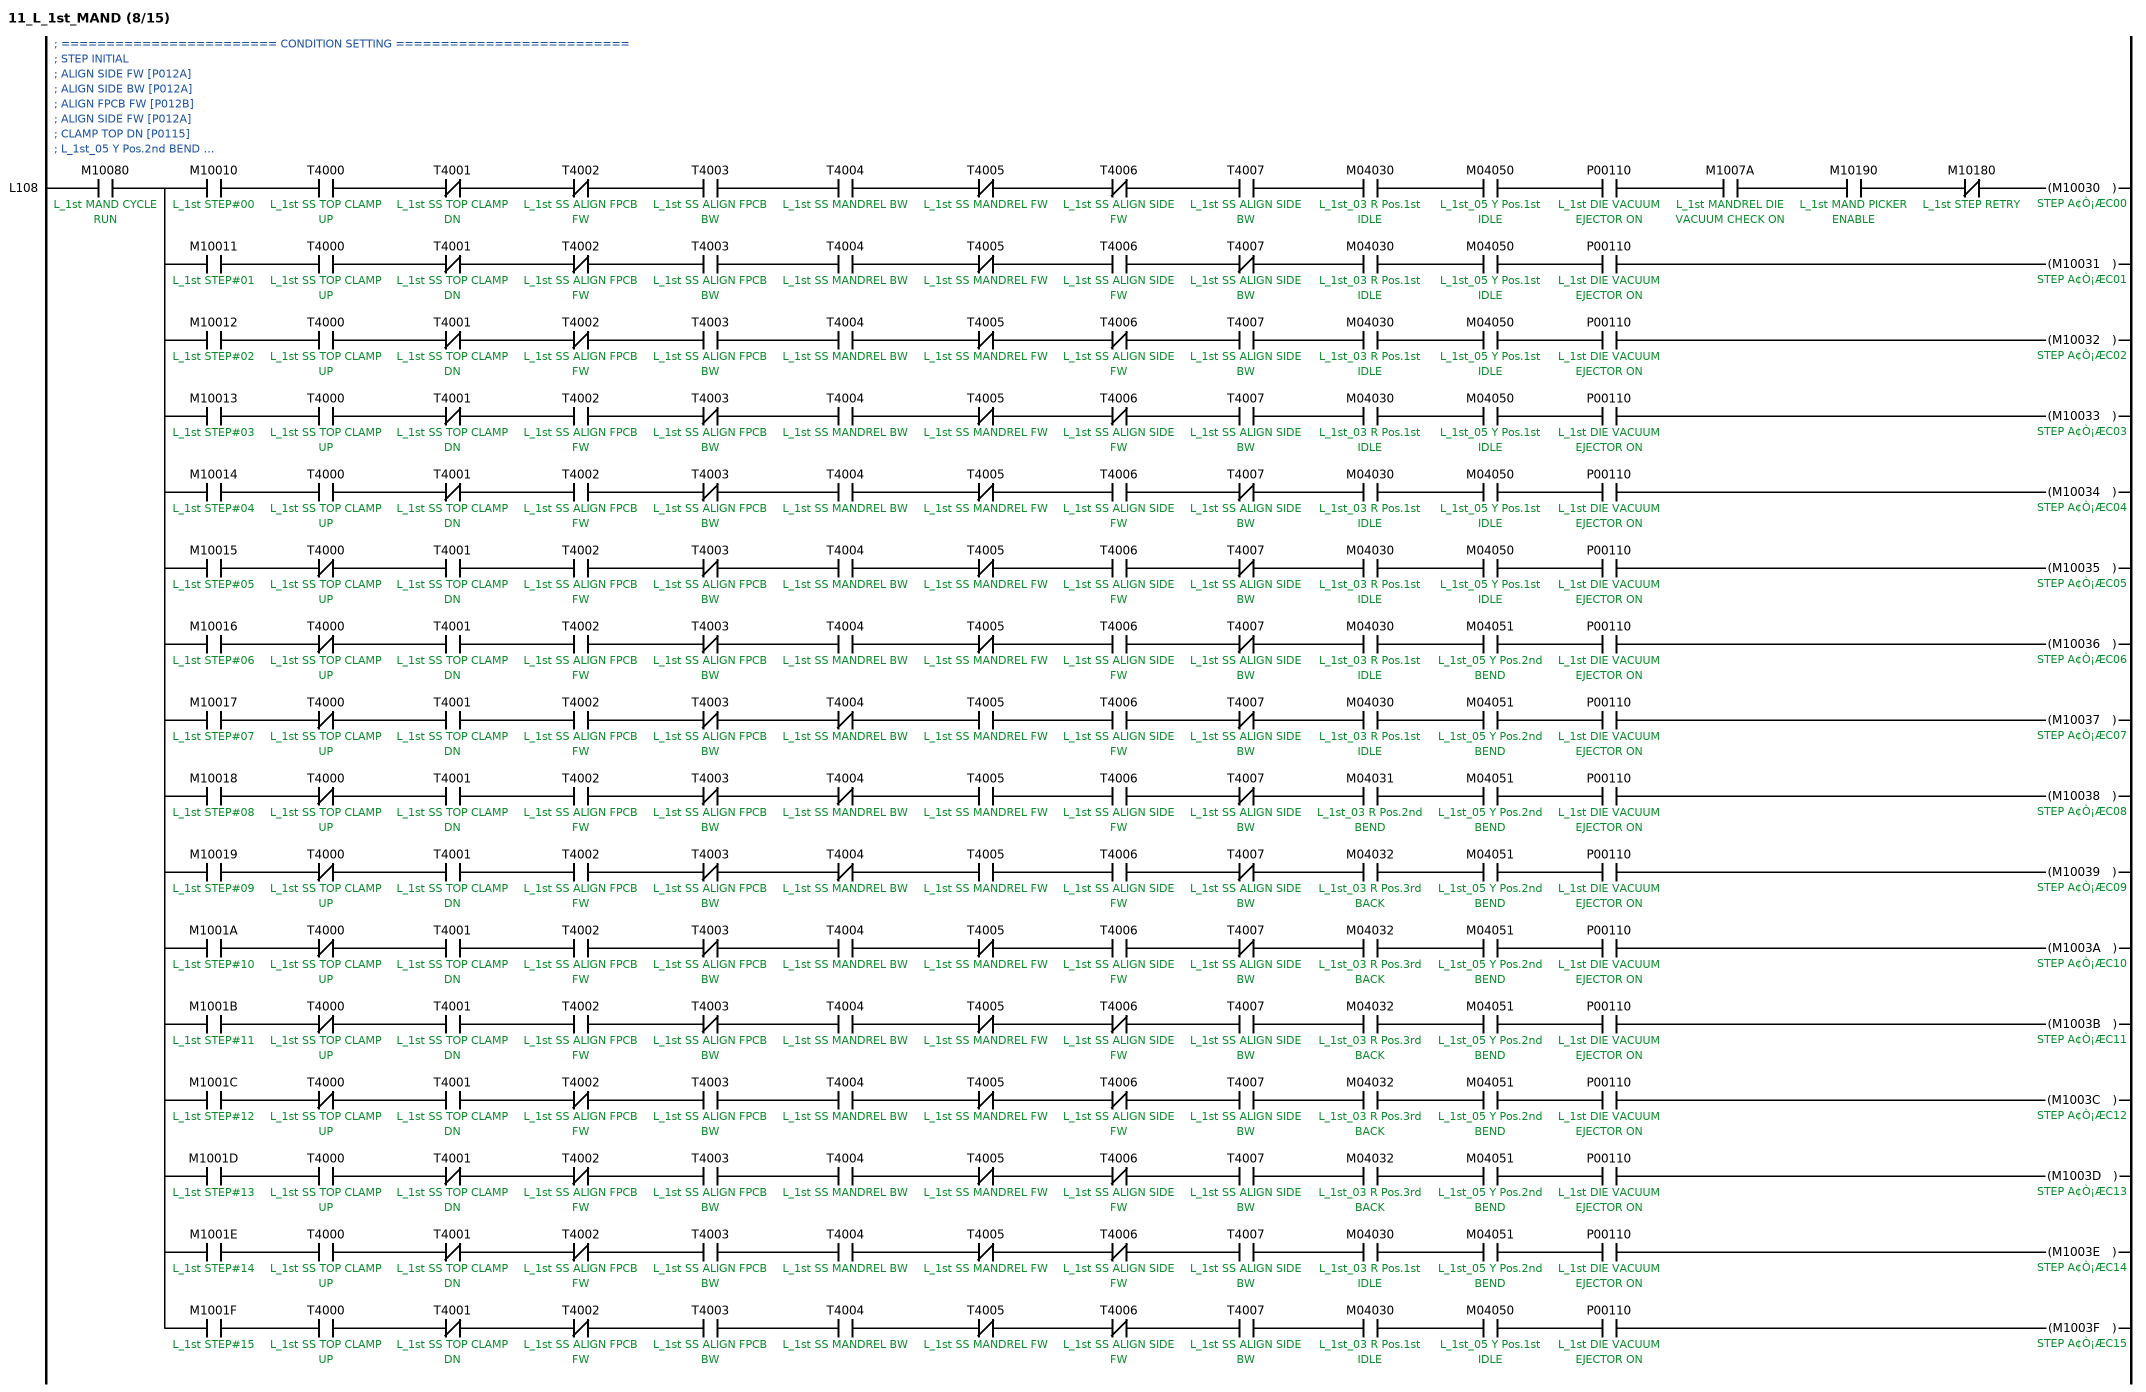
// ======================== CONDITION SETTING ==========================
; L108
LOAD      M10080	// L_1st MAND CYCLE RUN
MPUSH
AND       M10010	// L_1st STEP#00
AND       T4000	// L_1st SS TOP CLAMP    UP
AND NOT   T4001	// L_1st SS TOP CLAMP    DN
AND NOT   T4002	// L_1st SS ALIGN FPCB FW
AND       T4003	// L_1st SS ALIGN FPCB BW
AND       T4004	// L_1st SS MANDREL BW
AND NOT   T4005	// L_1st SS MANDREL FW
AND NOT   T4006	// L_1st SS ALIGN SIDE FW
AND       T4007	// L_1st SS ALIGN SIDE BW
AND       M04030	// L_1st_03 R Pos.1st IDLE
AND       M04050	// L_1st_05 Y Pos.1st IDLE
AND       P00110	// L_1st DIE VACUUM EJECTOR ON
AND       M1007A	// L_1st MANDREL DIE VACUUM CHECK ON
AND       M10190	// L_1st MAND PICKER ENABLE
AND NOT   M10180	// L_1st STEP RETRY
OUT       M10030	// STEP A¢Ò¡ÆC00
MLOAD
AND       M10011	// L_1st STEP#01
AND       T4000	// L_1st SS TOP CLAMP    UP
AND NOT   T4001	// L_1st SS TOP CLAMP    DN
AND NOT   T4002	// L_1st SS ALIGN FPCB FW
AND       T4003	// L_1st SS ALIGN FPCB BW
AND       T4004	// L_1st SS MANDREL BW
AND NOT   T4005	// L_1st SS MANDREL FW
AND       T4006	// L_1st SS ALIGN SIDE FW
AND NOT   T4007	// L_1st SS ALIGN SIDE BW
AND       M04030	// L_1st_03 R Pos.1st IDLE
AND       M04050	// L_1st_05 Y Pos.1st IDLE
AND       P00110	// L_1st DIE VACUUM EJECTOR ON
OUT       M10031	// STEP A¢Ò¡ÆC01
MLOAD
AND       M10012	// L_1st STEP#02
AND       T4000	// L_1st SS TOP CLAMP    UP
AND NOT   T4001	// L_1st SS TOP CLAMP    DN
AND NOT   T4002	// L_1st SS ALIGN FPCB FW
AND       T4003	// L_1st SS ALIGN FPCB BW
AND       T4004	// L_1st SS MANDREL BW
AND NOT   T4005	// L_1st SS MANDREL FW
AND NOT   T4006	// L_1st SS ALIGN SIDE FW
AND       T4007	// L_1st SS ALIGN SIDE BW
AND       M04030	// L_1st_03 R Pos.1st IDLE
AND       M04050	// L_1st_05 Y Pos.1st IDLE
AND       P00110	// L_1st DIE VACUUM EJECTOR ON
OUT       M10032	// STEP A¢Ò¡ÆC02
MLOAD
AND       M10013	// L_1st STEP#03
AND       T4000	// L_1st SS TOP CLAMP    UP
AND NOT   T4001	// L_1st SS TOP CLAMP    DN
AND       T4002	// L_1st SS ALIGN FPCB FW
AND NOT   T4003	// L_1st SS ALIGN FPCB BW
AND       T4004	// L_1st SS MANDREL BW
AND NOT   T4005	// L_1st SS MANDREL FW
AND NOT   T4006	// L_1st SS ALIGN SIDE FW
AND       T4007	// L_1st SS ALIGN SIDE BW
AND       M04030	// L_1st_03 R Pos.1st IDLE
AND       M04050	// L_1st_05 Y Pos.1st IDLE
AND       P00110	// L_1st DIE VACUUM EJECTOR ON
OUT       M10033	// STEP A¢Ò¡ÆC03
MLOAD
AND       M10014	// L_1st STEP#04
AND       T4000	// L_1st SS TOP CLAMP    UP
AND NOT   T4001	// L_1st SS TOP CLAMP    DN
AND       T4002	// L_1st SS ALIGN FPCB FW
AND NOT   T4003	// L_1st SS ALIGN FPCB BW
AND       T4004	// L_1st SS MANDREL BW
AND NOT   T4005	// L_1st SS MANDREL FW
AND       T4006	// L_1st SS ALIGN SIDE FW
AND NOT   T4007	// L_1st SS ALIGN SIDE BW
AND       M04030	// L_1st_03 R Pos.1st IDLE
AND       M04050	// L_1st_05 Y Pos.1st IDLE
AND       P00110	// L_1st DIE VACUUM EJECTOR ON
OUT       M10034	// STEP A¢Ò¡ÆC04
MLOAD
AND       M10015	// L_1st STEP#05
AND NOT   T4000	// L_1st SS TOP CLAMP    UP
AND       T4001	// L_1st SS TOP CLAMP    DN
AND       T4002	// L_1st SS ALIGN FPCB FW
AND NOT   T4003	// L_1st SS ALIGN FPCB BW
AND       T4004	// L_1st SS MANDREL BW
AND NOT   T4005	// L_1st SS MANDREL FW
AND       T4006	// L_1st SS ALIGN SIDE FW
AND NOT   T4007	// L_1st SS ALIGN SIDE BW
AND       M04030	// L_1st_03 R Pos.1st IDLE
AND       M04050	// L_1st_05 Y Pos.1st IDLE
AND       P00110	// L_1st DIE VACUUM EJECTOR ON
OUT       M10035	// STEP A¢Ò¡ÆC05
MLOAD
AND       M10016	// L_1st STEP#06
AND NOT   T4000	// L_1st SS TOP CLAMP    UP
AND       T4001	// L_1st SS TOP CLAMP    DN
AND       T4002	// L_1st SS ALIGN FPCB FW
AND NOT   T4003	// L_1st SS ALIGN FPCB BW
AND       T4004	// L_1st SS MANDREL BW
AND NOT   T4005	// L_1st SS MANDREL FW
AND       T4006	// L_1st SS ALIGN SIDE FW
AND NOT   T4007	// L_1st SS ALIGN SIDE BW
AND       M04030	// L_1st_03 R Pos.1st IDLE
AND       M04051	// L_1st_05 Y Pos.2nd BEND
AND       P00110	// L_1st DIE VACUUM EJECTOR ON
OUT       M10036	// STEP A¢Ò¡ÆC06
MLOAD
AND       M10017	// L_1st STEP#07
AND NOT   T4000	// L_1st SS TOP CLAMP    UP
AND       T4001	// L_1st SS TOP CLAMP    DN
AND       T4002	// L_1st SS ALIGN FPCB FW
AND NOT   T4003	// L_1st SS ALIGN FPCB BW
AND NOT   T4004	// L_1st SS MANDREL BW
AND       T4005	// L_1st SS MANDREL FW
AND       T4006	// L_1st SS ALIGN SIDE FW
AND NOT   T4007	// L_1st SS ALIGN SIDE BW
AND       M04030	// L_1st_03 R Pos.1st IDLE
AND       M04051	// L_1st_05 Y Pos.2nd BEND
AND       P00110	// L_1st DIE VACUUM EJECTOR ON
OUT       M10037	// STEP A¢Ò¡ÆC07
MLOAD
AND       M10018	// L_1st STEP#08
AND NOT   T4000	// L_1st SS TOP CLAMP    UP
AND       T4001	// L_1st SS TOP CLAMP    DN
AND       T4002	// L_1st SS ALIGN FPCB FW
AND NOT   T4003	// L_1st SS ALIGN FPCB BW
AND NOT   T4004	// L_1st SS MANDREL BW
AND       T4005	// L_1st SS MANDREL FW
AND       T4006	// L_1st SS ALIGN SIDE FW
AND NOT   T4007	// L_1st SS ALIGN SIDE BW
AND       M04031	// L_1st_03 R Pos.2nd BEND
AND       M04051	// L_1st_05 Y Pos.2nd BEND
AND       P00110	// L_1st DIE VACUUM EJECTOR ON
OUT       M10038	// STEP A¢Ò¡ÆC08
MLOAD
AND       M10019	// L_1st STEP#09
AND NOT   T4000	// L_1st SS TOP CLAMP    UP
AND       T4001	// L_1st SS TOP CLAMP    DN
AND       T4002	// L_1st SS ALIGN FPCB FW
AND NOT   T4003	// L_1st SS ALIGN FPCB BW
AND NOT   T4004	// L_1st SS MANDREL BW
AND       T4005	// L_1st SS MANDREL FW
AND       T4006	// L_1st SS ALIGN SIDE FW
AND NOT   T4007	// L_1st SS ALIGN SIDE BW
AND       M04032	// L_1st_03 R Pos.3rd BACK
AND       M04051	// L_1st_05 Y Pos.2nd BEND
AND       P00110	// L_1st DIE VACUUM EJECTOR ON
OUT       M10039	// STEP A¢Ò¡ÆC09
MLOAD
AND       M1001A	// L_1st STEP#10
AND NOT   T4000	// L_1st SS TOP CLAMP    UP
AND       T4001	// L_1st SS TOP CLAMP    DN
AND       T4002	// L_1st SS ALIGN FPCB FW
AND NOT   T4003	// L_1st SS ALIGN FPCB BW
AND       T4004	// L_1st SS MANDREL BW
AND NOT   T4005	// L_1st SS MANDREL FW
AND       T4006	// L_1st SS ALIGN SIDE FW
AND NOT   T4007	// L_1st SS ALIGN SIDE BW
AND       M04032	// L_1st_03 R Pos.3rd BACK
AND       M04051	// L_1st_05 Y Pos.2nd BEND
AND       P00110	// L_1st DIE VACUUM EJECTOR ON
OUT       M1003A	// STEP A¢Ò¡ÆC10
MLOAD
AND       M1001B	// L_1st STEP#11
AND NOT   T4000	// L_1st SS TOP CLAMP    UP
AND       T4001	// L_1st SS TOP CLAMP    DN
AND       T4002	// L_1st SS ALIGN FPCB FW
AND NOT   T4003	// L_1st SS ALIGN FPCB BW
AND       T4004	// L_1st SS MANDREL BW
AND NOT   T4005	// L_1st SS MANDREL FW
AND NOT   T4006	// L_1st SS ALIGN SIDE FW
AND       T4007	// L_1st SS ALIGN SIDE BW
AND       M04032	// L_1st_03 R Pos.3rd BACK
AND       M04051	// L_1st_05 Y Pos.2nd BEND
AND       P00110	// L_1st DIE VACUUM EJECTOR ON
OUT       M1003B	// STEP A¢Ò¡ÆC11
MLOAD
AND       M1001C	// L_1st STEP#12
AND NOT   T4000	// L_1st SS TOP CLAMP    UP
AND       T4001	// L_1st SS TOP CLAMP    DN
AND NOT   T4002	// L_1st SS ALIGN FPCB FW
AND       T4003	// L_1st SS ALIGN FPCB BW
AND       T4004	// L_1st SS MANDREL BW
AND NOT   T4005	// L_1st SS MANDREL FW
AND NOT   T4006	// L_1st SS ALIGN SIDE FW
AND       T4007	// L_1st SS ALIGN SIDE BW
AND       M04032	// L_1st_03 R Pos.3rd BACK
AND       M04051	// L_1st_05 Y Pos.2nd BEND
AND       P00110	// L_1st DIE VACUUM EJECTOR ON
OUT       M1003C	// STEP A¢Ò¡ÆC12
MLOAD
AND       M1001D	// L_1st STEP#13
AND       T4000	// L_1st SS TOP CLAMP    UP
AND NOT   T4001	// L_1st SS TOP CLAMP    DN
AND NOT   T4002	// L_1st SS ALIGN FPCB FW
AND       T4003	// L_1st SS ALIGN FPCB BW
AND       T4004	// L_1st SS MANDREL BW
AND NOT   T4005	// L_1st SS MANDREL FW
AND NOT   T4006	// L_1st SS ALIGN SIDE FW
AND       T4007	// L_1st SS ALIGN SIDE BW
AND       M04032	// L_1st_03 R Pos.3rd BACK
AND       M04051	// L_1st_05 Y Pos.2nd BEND
AND       P00110	// L_1st DIE VACUUM EJECTOR ON
OUT       M1003D	// STEP A¢Ò¡ÆC13
MLOAD
AND       M1001E	// L_1st STEP#14
AND       T4000	// L_1st SS TOP CLAMP    UP
AND NOT   T4001	// L_1st SS TOP CLAMP    DN
AND NOT   T4002	// L_1st SS ALIGN FPCB FW
AND       T4003	// L_1st SS ALIGN FPCB BW
AND       T4004	// L_1st SS MANDREL BW
AND NOT   T4005	// L_1st SS MANDREL FW
AND NOT   T4006	// L_1st SS ALIGN SIDE FW
AND       T4007	// L_1st SS ALIGN SIDE BW
AND       M04030	// L_1st_03 R Pos.1st IDLE
AND       M04051	// L_1st_05 Y Pos.2nd BEND
AND       P00110	// L_1st DIE VACUUM EJECTOR ON
OUT       M1003E	// STEP A¢Ò¡ÆC14
MPOP
AND       M1001F	// L_1st STEP#15
AND       T4000	// L_1st SS TOP CLAMP    UP
AND NOT   T4001	// L_1st SS TOP CLAMP    DN
AND NOT   T4002	// L_1st SS ALIGN FPCB FW
AND       T4003	// L_1st SS ALIGN FPCB BW
AND       T4004	// L_1st SS MANDREL BW
AND NOT   T4005	// L_1st SS MANDREL FW
AND NOT   T4006	// L_1st SS ALIGN SIDE FW
AND       T4007	// L_1st SS ALIGN SIDE BW
AND       M04030	// L_1st_03 R Pos.1st IDLE
AND       M04050	// L_1st_05 Y Pos.1st IDLE
AND       P00110	// L_1st DIE VACUUM EJECTOR ON
OUT       M1003F	// STEP A¢Ò¡ÆC15
// output comment: STEP INITIAL
// output comment: ALIGN SIDE FW [P012A]
// output comment: ALIGN SIDE BW [P012A]
// output comment: ALIGN FPCB FW [P012B]
// output comment: ALIGN SIDE FW [P012A]
// output comment: CLAMP TOP DN [P0115]
// output comment: L_1st_05 Y Pos.2nd BEND >
// output comment: MANDREL FW    [P0114]
// output comment: L_1st_03 R Pos.2nd BEND >
// output comment: L_1st_03 R Pos.3rd BACK >
// output comment: MANDREL BW    [P0114]
// output comment: ALIGN SIDE BW [P012A]
// output comment: ALIGN FPCB BW [P012B]
// output comment: CLAMP TOP UP [P0115]
// output comment: L_1st_03 R Pos.1st IDLE >
// output comment: L_1st_05 Y Pos.1st IDLE >

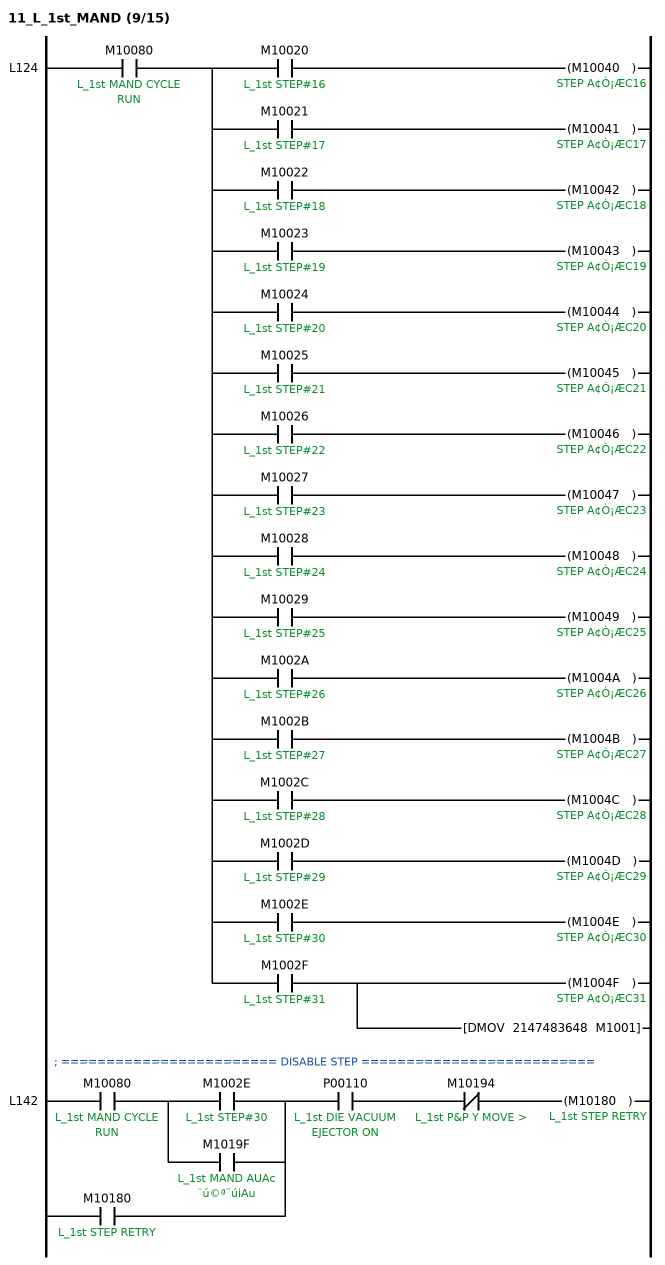
; L124
LOAD      M10080	// L_1st MAND CYCLE RUN
MPUSH
AND       M10020	// L_1st STEP#16
OUT       M10040	// STEP A¢Ò¡ÆC16
MLOAD
AND       M10021	// L_1st STEP#17
OUT       M10041	// STEP A¢Ò¡ÆC17
MLOAD
AND       M10022	// L_1st STEP#18
OUT       M10042	// STEP A¢Ò¡ÆC18
MLOAD
AND       M10023	// L_1st STEP#19
OUT       M10043	// STEP A¢Ò¡ÆC19
MLOAD
AND       M10024	// L_1st STEP#20
OUT       M10044	// STEP A¢Ò¡ÆC20
MLOAD
AND       M10025	// L_1st STEP#21
OUT       M10045	// STEP A¢Ò¡ÆC21
MLOAD
AND       M10026	// L_1st STEP#22
OUT       M10046	// STEP A¢Ò¡ÆC22
MLOAD
AND       M10027	// L_1st STEP#23
OUT       M10047	// STEP A¢Ò¡ÆC23
MLOAD
AND       M10028	// L_1st STEP#24
OUT       M10048	// STEP A¢Ò¡ÆC24
MLOAD
AND       M10029	// L_1st STEP#25
OUT       M10049	// STEP A¢Ò¡ÆC25
MLOAD
AND       M1002A	// L_1st STEP#26
OUT       M1004A	// STEP A¢Ò¡ÆC26
MLOAD
AND       M1002B	// L_1st STEP#27
OUT       M1004B	// STEP A¢Ò¡ÆC27
MLOAD
AND       M1002C	// L_1st STEP#28
OUT       M1004C	// STEP A¢Ò¡ÆC28
MLOAD
AND       M1002D	// L_1st STEP#29
OUT       M1004D	// STEP A¢Ò¡ÆC29
MLOAD
AND       M1002E	// L_1st STEP#30
OUT       M1004E	// STEP A¢Ò¡ÆC30
MPOP
AND       M1002F	// L_1st STEP#31
OUT       M1004F	// STEP A¢Ò¡ÆC31
DMOV      2147483648 M1001
// ======================== DISABLE STEP ==========================
; L142
LOAD      M10080	// L_1st MAND CYCLE RUN
LOAD      M1002E	// L_1st STEP#30
OR        M1019F	// L_1st MAND AUAc ¨ú©ª¨úiAu
AND LOAD
OR        M10180	// L_1st STEP RETRY
AND       P00110	// L_1st DIE VACUUM EJECTOR ON
AND NOT   M10194	// L_1st P&P Y MOVE >
OUT       M10180	// L_1st STEP RETRY

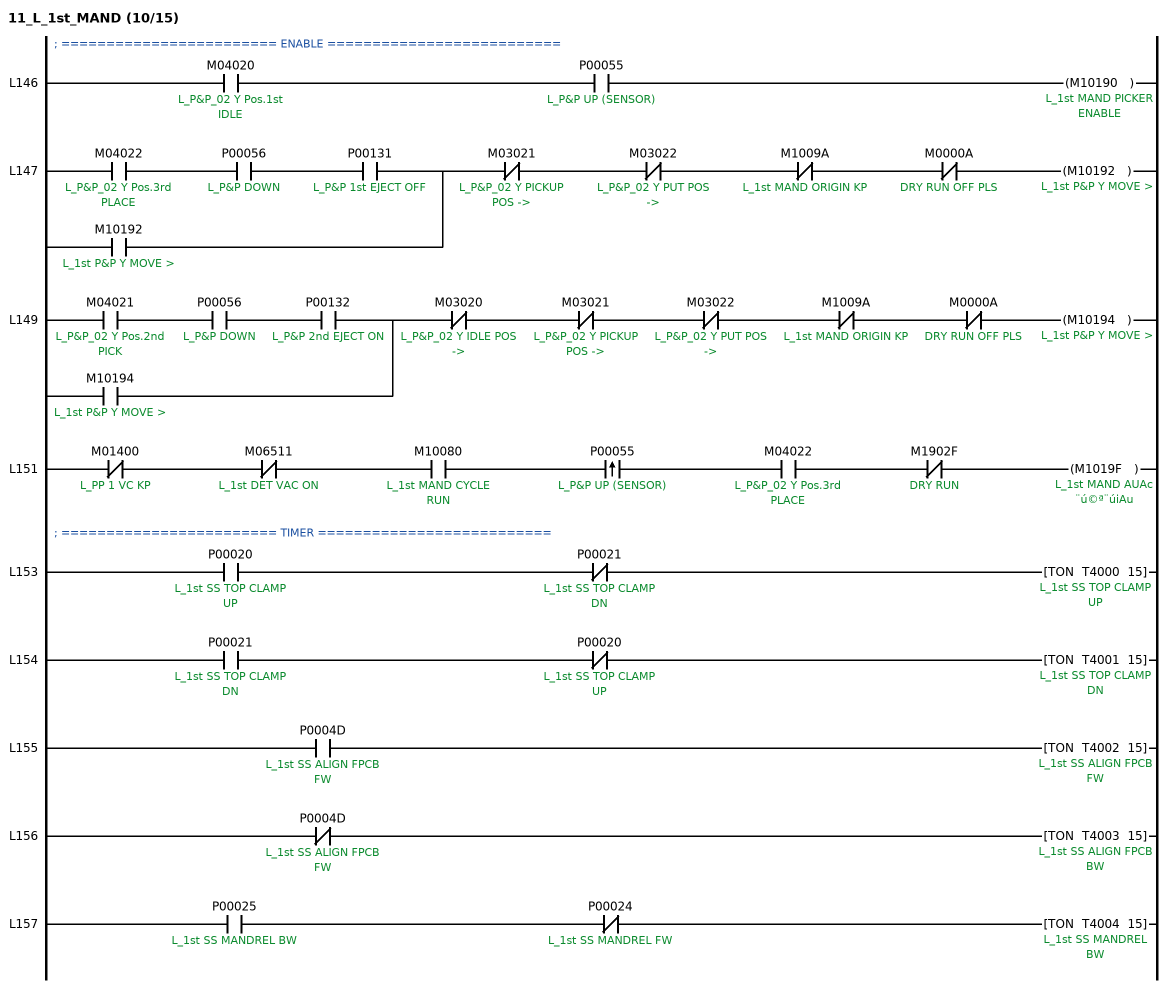
// ======================== ENABLE ==========================
; L146
LOAD      M04020	// L_P&P_02 Y Pos.1st IDLE
AND       P00055	// L_P&P UP (SENSOR)
OUT       M10190	// L_1st MAND PICKER ENABLE
; L147
LOAD      M04022	// L_P&P_02 Y Pos.3rd PLACE
AND       P00056	// L_P&P DOWN
AND       P00131	// L_P&P 1st EJECT OFF
OR        M10192	// L_1st P&P Y MOVE >
AND NOT   M03021	// L_P&P_02 Y PICKUP POS ->
AND NOT   M03022	// L_P&P_02 Y PUT POS ->
AND NOT   M1009A	// L_1st MAND ORIGIN KP
AND NOT   M0000A	// DRY RUN OFF PLS
OUT       M10192	// L_1st P&P Y MOVE >
; L149
LOAD      M04021	// L_P&P_02 Y Pos.2nd PICK
AND       P00056	// L_P&P DOWN
AND       P00132	// L_P&P 2nd EJECT ON
OR        M10194	// L_1st P&P Y MOVE >
AND NOT   M03020	// L_P&P_02 Y IDLE POS ->
AND NOT   M03021	// L_P&P_02 Y PICKUP POS ->
AND NOT   M03022	// L_P&P_02 Y PUT POS ->
AND NOT   M1009A	// L_1st MAND ORIGIN KP
AND NOT   M0000A	// DRY RUN OFF PLS
OUT       M10194	// L_1st P&P Y MOVE >
; L151
LOAD NOT  M01400	// L_PP 1 VC KP
AND NOT   M06511	// L_1st DET VAC ON
AND       M10080	// L_1st MAND CYCLE RUN
ANDP      P00055	// L_P&P UP (SENSOR)
AND       M04022	// L_P&P_02 Y Pos.3rd PLACE
AND NOT   M1902F	// DRY RUN
OUT       M1019F	// L_1st MAND AUAc ¨ú©ª¨úiAu
// ======================== TIMER ==========================
; L153
LOAD      P00020	// L_1st SS TOP CLAMP UP
AND NOT   P00021	// L_1st SS TOP CLAMP DN
TON       T4000 15	// L_1st SS TOP CLAMP    UP
; L154
LOAD      P00021	// L_1st SS TOP CLAMP DN
AND NOT   P00020	// L_1st SS TOP CLAMP UP
TON       T4001 15	// L_1st SS TOP CLAMP    DN
; L155
LOAD      P0004D	// L_1st SS ALIGN FPCB FW
TON       T4002 15	// L_1st SS ALIGN FPCB FW
; L156
LOAD NOT  P0004D	// L_1st SS ALIGN FPCB FW
TON       T4003 15	// L_1st SS ALIGN FPCB BW
; L157
LOAD      P00025	// L_1st SS MANDREL BW
AND NOT   P00024	// L_1st SS MANDREL FW
TON       T4004 15	// L_1st SS MANDREL BW

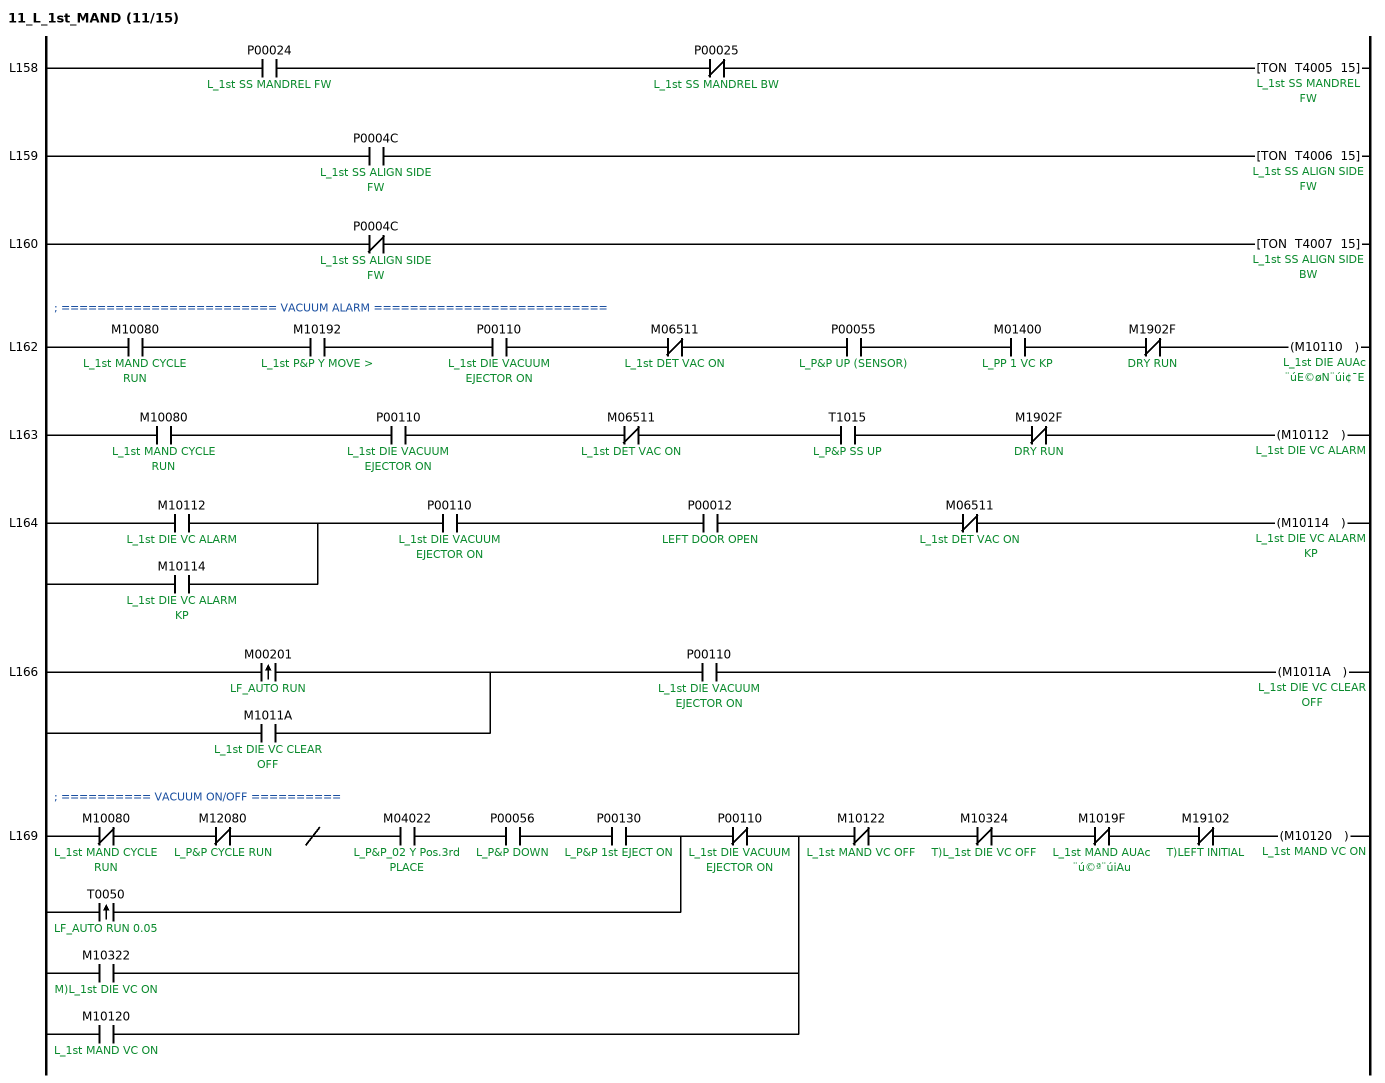
; L158
LOAD      P00024	// L_1st SS MANDREL FW
AND NOT   P00025	// L_1st SS MANDREL BW
TON       T4005 15	// L_1st SS MANDREL FW
; L159
LOAD      P0004C	// L_1st SS ALIGN SIDE FW
TON       T4006 15	// L_1st SS ALIGN SIDE FW
; L160
LOAD NOT  P0004C	// L_1st SS ALIGN SIDE FW
TON       T4007 15	// L_1st SS ALIGN SIDE BW
// ======================== VACUUM ALARM ==========================
; L162
LOAD      M10080	// L_1st MAND CYCLE RUN
AND       M10192	// L_1st P&P Y MOVE >
AND       P00110	// L_1st DIE VACUUM EJECTOR ON
AND NOT   M06511	// L_1st DET VAC ON
AND       P00055	// L_P&P UP (SENSOR)
AND       M01400	// L_PP 1 VC KP
AND NOT   M1902F	// DRY RUN
OUT       M10110	// L_1st DIE AUAc ¨úE©øN¨úi¢¯E
; L163
LOAD      M10080	// L_1st MAND CYCLE RUN
AND       P00110	// L_1st DIE VACUUM EJECTOR ON
AND NOT   M06511	// L_1st DET VAC ON
AND       T1015	// L_P&P SS UP
AND NOT   M1902F	// DRY RUN
OUT       M10112	// L_1st DIE VC ALARM
; L164
LOAD      M10112	// L_1st DIE VC ALARM
OR        M10114	// L_1st DIE VC ALARM KP
AND       P00110	// L_1st DIE VACUUM EJECTOR ON
AND       P00012	// LEFT DOOR OPEN
AND NOT   M06511	// L_1st DET VAC ON
OUT       M10114	// L_1st DIE VC ALARM KP
; L166
LOADP     M00201	// LF_AUTO RUN
OR        M1011A	// L_1st DIE VC CLEAR OFF
AND       P00110	// L_1st DIE VACUUM EJECTOR ON
OUT       M1011A	// L_1st DIE VC CLEAR OFF
// ========== VACUUM ON/OFF ==========
; L169
LOAD NOT  M10080	// L_1st MAND CYCLE RUN
AND NOT   M12080	// L_P&P CYCLE RUN
NOT
AND       M04022	// L_P&P_02 Y Pos.3rd PLACE
AND       P00056	// L_P&P DOWN
AND       P00130	// L_P&P 1st EJECT ON
ORP       T0050	// LF_AUTO RUN 0.05
AND NOT   P00110	// L_1st DIE VACUUM EJECTOR ON
OR        M10322	// M)L_1st DIE VC ON
OR        M10120	// L_1st MAND VC ON
AND NOT   M10122	// L_1st MAND VC OFF
AND NOT   M10324	// T)L_1st DIE VC OFF
AND NOT   M1019F	// L_1st MAND AUAc ¨ú©ª¨úiAu
AND NOT   M19102	// T)LEFT INITIAL
OUT       M10120	// L_1st MAND VC ON

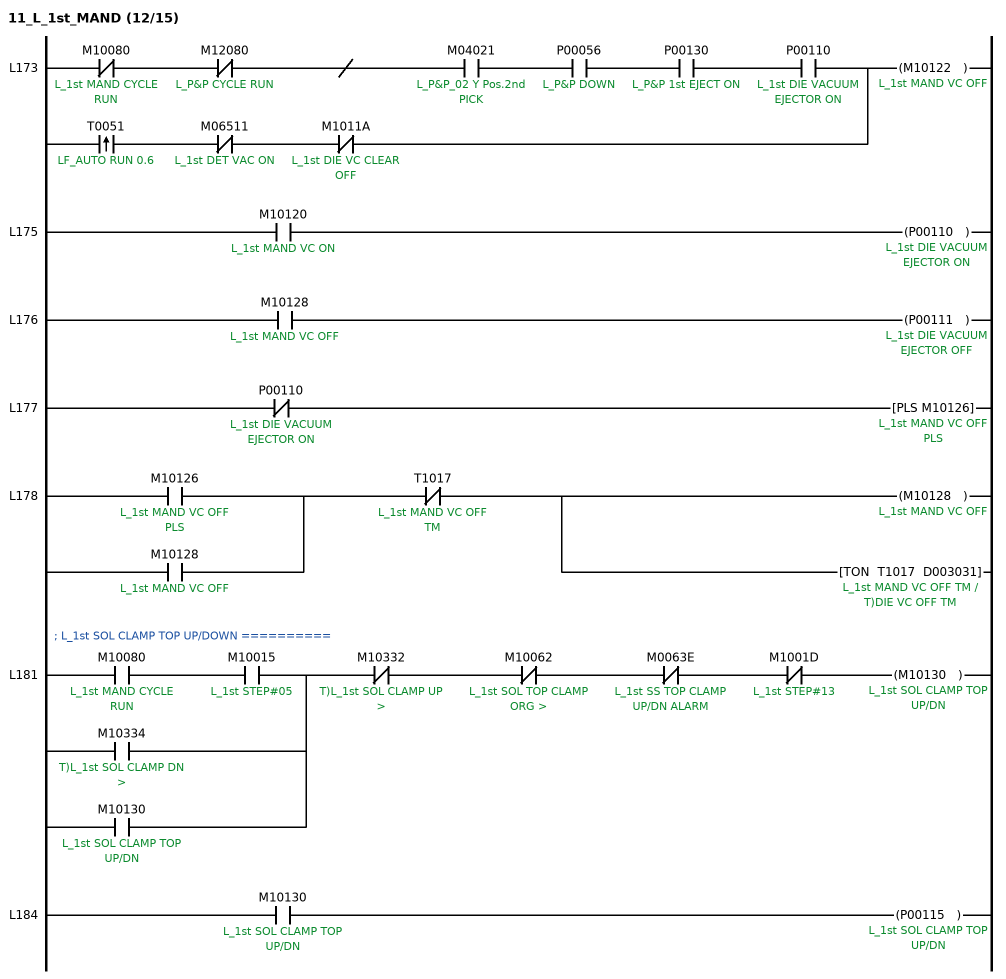
; L173
LOAD NOT  M10080	// L_1st MAND CYCLE RUN
AND NOT   M12080	// L_P&P CYCLE RUN
NOT
AND       M04021	// L_P&P_02 Y Pos.2nd PICK
AND       P00056	// L_P&P DOWN
AND       P00130	// L_P&P 1st EJECT ON
AND       P00110	// L_1st DIE VACUUM EJECTOR ON
LOADP     T0051	// LF_AUTO RUN 0.6
AND NOT   M06511	// L_1st DET VAC ON
AND NOT   M1011A	// L_1st DIE VC CLEAR OFF
OR LOAD
OUT       M10122	// L_1st MAND VC OFF
; L175
LOAD      M10120	// L_1st MAND VC ON
OUT       P00110	// L_1st DIE VACUUM EJECTOR ON
; L176
LOAD      M10128	// L_1st MAND VC OFF
OUT       P00111	// L_1st DIE VACUUM EJECTOR OFF
; L177
LOAD NOT  P00110	// L_1st DIE VACUUM EJECTOR ON
OUTP      M10126	// L_1st MAND VC OFF PLS
; L178
LOAD      M10126	// L_1st MAND VC OFF PLS
OR        M10128	// L_1st MAND VC OFF
AND NOT   T1017	// L_1st MAND VC OFF TM
OUT       M10128	// L_1st MAND VC OFF
TON       T1017 D003031	// L_1st MAND VC OFF TM / T)DIE VC OFF TM
// L_1st SOL CLAMP TOP UP/DOWN ==========
; L181
LOAD      M10080	// L_1st MAND CYCLE RUN
AND       M10015	// L_1st STEP#05
OR        M10334	// T)L_1st SOL CLAMP DN >
OR        M10130	// L_1st SOL CLAMP TOP UP/DN
AND NOT   M10332	// T)L_1st SOL CLAMP UP >
AND NOT   M10062	// L_1st SOL TOP CLAMP ORG >
AND NOT   M0063E	// L_1st SS TOP CLAMP UP/DN ALARM
AND NOT   M1001D	// L_1st STEP#13
OUT       M10130	// L_1st SOL CLAMP TOP UP/DN
; L184
LOAD      M10130	// L_1st SOL CLAMP TOP UP/DN
OUT       P00115	// L_1st SOL CLAMP TOP UP/DN

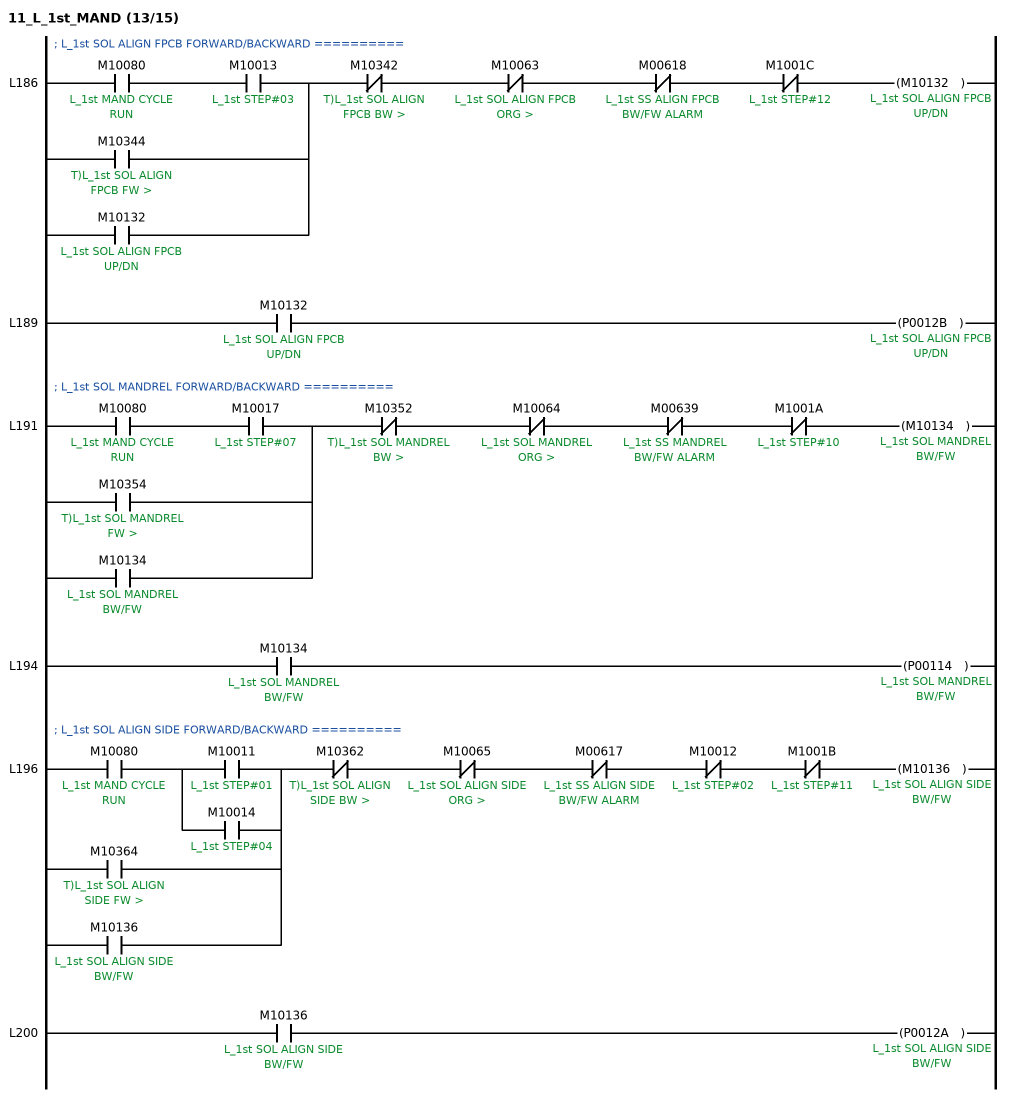
// L_1st SOL ALIGN FPCB FORWARD/BACKWARD ==========
; L186
LOAD      M10080	// L_1st MAND CYCLE RUN
AND       M10013	// L_1st STEP#03
OR        M10344	// T)L_1st SOL ALIGN FPCB FW >
OR        M10132	// L_1st SOL ALIGN FPCB UP/DN
AND NOT   M10342	// T)L_1st SOL ALIGN FPCB BW >
AND NOT   M10063	// L_1st SOL ALIGN FPCB ORG >
AND NOT   M00618	// L_1st SS ALIGN FPCB BW/FW ALARM
AND NOT   M1001C	// L_1st STEP#12
OUT       M10132	// L_1st SOL ALIGN FPCB UP/DN
; L189
LOAD      M10132	// L_1st SOL ALIGN FPCB UP/DN
OUT       P0012B	// L_1st SOL ALIGN FPCB UP/DN
// L_1st SOL MANDREL FORWARD/BACKWARD ==========
; L191
LOAD      M10080	// L_1st MAND CYCLE RUN
AND       M10017	// L_1st STEP#07
OR        M10354	// T)L_1st SOL MANDREL FW >
OR        M10134	// L_1st SOL MANDREL BW/FW
AND NOT   M10352	// T)L_1st SOL MANDREL BW >
AND NOT   M10064	// L_1st SOL MANDREL ORG >
AND NOT   M00639	// L_1st SS MANDREL BW/FW ALARM
AND NOT   M1001A	// L_1st STEP#10
OUT       M10134	// L_1st SOL MANDREL BW/FW
; L194
LOAD      M10134	// L_1st SOL MANDREL BW/FW
OUT       P00114	// L_1st SOL MANDREL BW/FW
// L_1st SOL ALIGN SIDE FORWARD/BACKWARD ==========
; L196
LOAD      M10080	// L_1st MAND CYCLE RUN
LOAD      M10011	// L_1st STEP#01
OR        M10014	// L_1st STEP#04
AND LOAD
OR        M10364	// T)L_1st SOL ALIGN SIDE FW >
OR        M10136	// L_1st SOL ALIGN SIDE BW/FW
AND NOT   M10362	// T)L_1st SOL ALIGN SIDE BW >
AND NOT   M10065	// L_1st SOL ALIGN SIDE ORG >
AND NOT   M00617	// L_1st SS ALIGN SIDE BW/FW ALARM
AND NOT   M10012	// L_1st STEP#02
AND NOT   M1001B	// L_1st STEP#11
OUT       M10136	// L_1st SOL ALIGN SIDE BW/FW
; L200
LOAD      M10136	// L_1st SOL ALIGN SIDE BW/FW
OUT       P0012A	// L_1st SOL ALIGN SIDE BW/FW

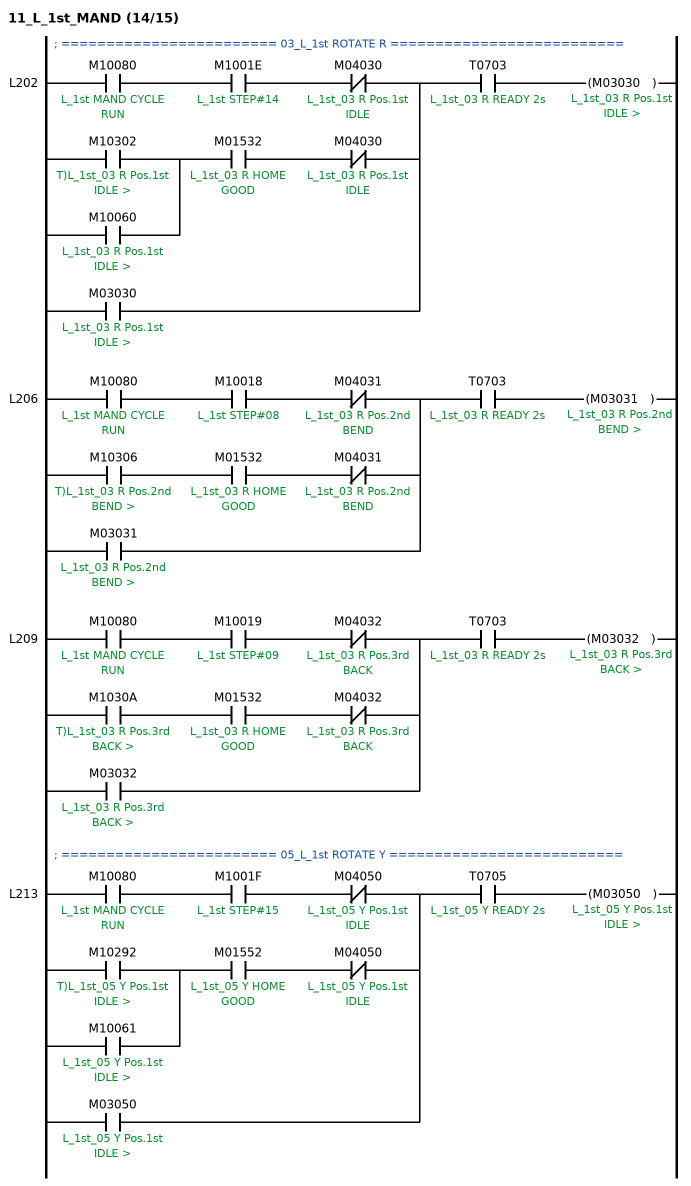
// ======================== 03_L_1st ROTATE R ==========================
; L202
LOAD      M10080	// L_1st MAND CYCLE RUN
AND       M1001E	// L_1st STEP#14
AND NOT   M04030	// L_1st_03 R Pos.1st IDLE
LOAD      M10302	// T)L_1st_03 R Pos.1st IDLE >
OR        M10060	// L_1st_03 R Pos.1st IDLE >
AND       M01532	// L_1st_03 R HOME GOOD
AND NOT   M04030	// L_1st_03 R Pos.1st IDLE
OR LOAD
OR        M03030	// L_1st_03 R Pos.1st IDLE >
AND       T0703	// L_1st_03 R READY 2s
OUT       M03030	// L_1st_03 R Pos.1st IDLE >
; L206
LOAD      M10080	// L_1st MAND CYCLE RUN
AND       M10018	// L_1st STEP#08
AND NOT   M04031	// L_1st_03 R Pos.2nd BEND
LOAD      M10306	// T)L_1st_03 R Pos.2nd BEND >
AND       M01532	// L_1st_03 R HOME GOOD
AND NOT   M04031	// L_1st_03 R Pos.2nd BEND
OR LOAD
OR        M03031	// L_1st_03 R Pos.2nd BEND >
AND       T0703	// L_1st_03 R READY 2s
OUT       M03031	// L_1st_03 R Pos.2nd BEND >
; L209
LOAD      M10080	// L_1st MAND CYCLE RUN
AND       M10019	// L_1st STEP#09
AND NOT   M04032	// L_1st_03 R Pos.3rd BACK
LOAD      M1030A	// T)L_1st_03 R Pos.3rd BACK >
AND       M01532	// L_1st_03 R HOME GOOD
AND NOT   M04032	// L_1st_03 R Pos.3rd BACK
OR LOAD
OR        M03032	// L_1st_03 R Pos.3rd BACK >
AND       T0703	// L_1st_03 R READY 2s
OUT       M03032	// L_1st_03 R Pos.3rd BACK >
// ======================== 05_L_1st ROTATE Y ==========================
; L213
LOAD      M10080	// L_1st MAND CYCLE RUN
AND       M1001F	// L_1st STEP#15
AND NOT   M04050	// L_1st_05 Y Pos.1st IDLE
LOAD      M10292	// T)L_1st_05 Y Pos.1st IDLE >
OR        M10061	// L_1st_05 Y Pos.1st IDLE >
AND       M01552	// L_1st_05 Y HOME GOOD
AND NOT   M04050	// L_1st_05 Y Pos.1st IDLE
OR LOAD
OR        M03050	// L_1st_05 Y Pos.1st IDLE >
AND       T0705	// L_1st_05 Y READY 2s
OUT       M03050	// L_1st_05 Y Pos.1st IDLE >

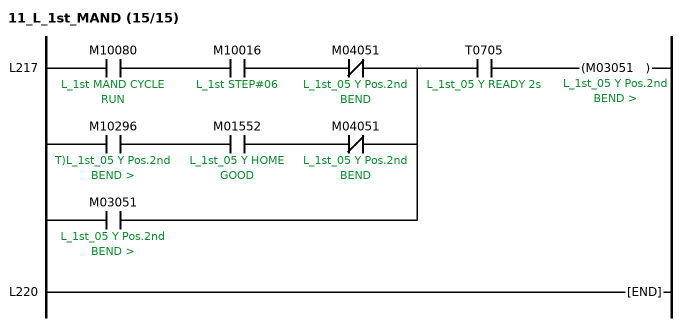
; L217
LOAD      M10080	// L_1st MAND CYCLE RUN
AND       M10016	// L_1st STEP#06
AND NOT   M04051	// L_1st_05 Y Pos.2nd BEND
LOAD      M10296	// T)L_1st_05 Y Pos.2nd BEND >
AND       M01552	// L_1st_05 Y HOME GOOD
AND NOT   M04051	// L_1st_05 Y Pos.2nd BEND
OR LOAD
OR        M03051	// L_1st_05 Y Pos.2nd BEND >
AND       T0705	// L_1st_05 Y READY 2s
OUT       M03051	// L_1st_05 Y Pos.2nd BEND >
; L220
END

PROGRAM 12_L_2nd_MAND (task: ¨ö¨¬A¥ì CA¡¤I¡¾¡¿¡¤¡Í)

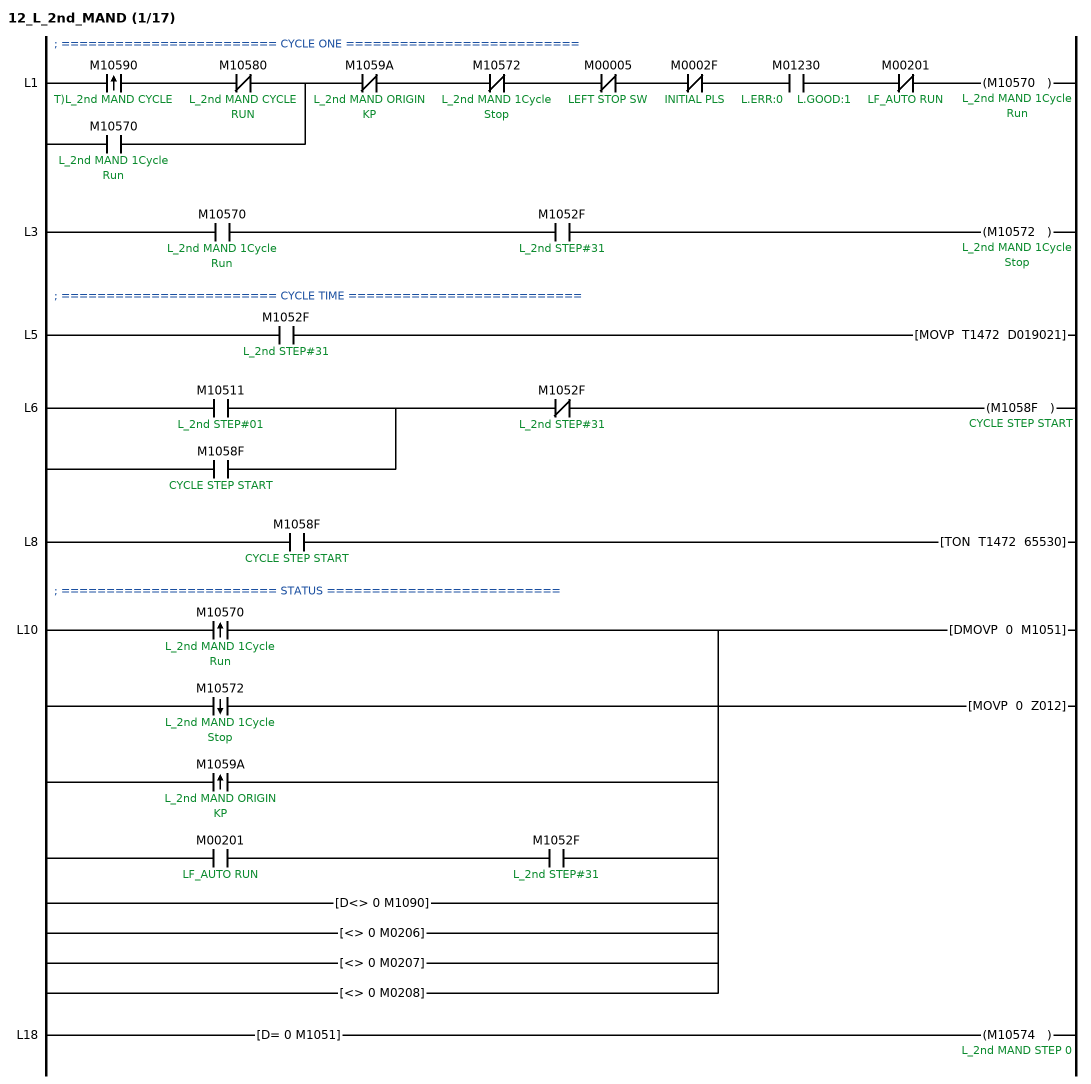
// ======================== CYCLE ONE ==========================
; L1
LOADP     M10590	// T)L_2nd MAND CYCLE
AND NOT   M10580	// L_2nd MAND CYCLE RUN
OR        M10570	// L_2nd MAND 1Cycle Run
AND NOT   M1059A	// L_2nd MAND ORIGIN KP
AND NOT   M10572	// L_2nd MAND 1Cycle Stop
AND NOT   M00005	// LEFT STOP SW
AND NOT   M0002F	// INITIAL PLS
AND       M01230	// L.ERR:0    L.GOOD:1
AND NOT   M00201	// LF_AUTO RUN
OUT       M10570	// L_2nd MAND 1Cycle Run
; L3
LOAD      M10570	// L_2nd MAND 1Cycle Run
AND       M1052F	// L_2nd STEP#31
OUT       M10572	// L_2nd MAND 1Cycle Stop
// ======================== CYCLE TIME ==========================
; L5
LOAD      M1052F	// L_2nd STEP#31
MOVP      T1472 D019021
; L6
LOAD      M10511	// L_2nd STEP#01
OR        M1058F	// CYCLE STEP START
AND NOT   M1052F	// L_2nd STEP#31
OUT       M1058F	// CYCLE STEP START
; L8
LOAD      M1058F	// CYCLE STEP START
TON       T1472 65530
// ======================== STATUS ==========================
; L10
LOADP     M10570	// L_2nd MAND 1Cycle Run
ORN       M10572	// L_2nd MAND 1Cycle Stop
ORP       M1059A	// L_2nd MAND ORIGIN KP
LOAD      M00201	// LF_AUTO RUN
AND       M1052F	// L_2nd STEP#31
OR LOAD
ORD<>     0 M1090
OR<>      0 M0206
OR<>      0 M0207
OR<>      0 M0208
DMOVP     0 M1051
MOVP      0 Z012
; L18
LOADD=    0 M1051
OUT       M10574	// L_2nd MAND STEP 0

